C03636=1129.592,11.692,-50.506,179.599,6.524,149.309
C03637=1129.598,11.442,-50.493,179.597,6.519,149.309
C03638=1129.621,10.298,-50.429,179.648,6.418,149.272
C03639=1129.626,10.070,-50.417,179.645,6.416,149.272
C03640=1129.630,9.842,-50.404,179.643,6.415,149.272
C03641=1129.635,9.614,-50.392,179.640,6.415,149.273
C03642=1129.640,9.364,-50.378,179.638,6.414,149.274
C03643=1129.645,9.115,-50.365,179.635,6.413,149.274
C03644=1129.651,8.864,-50.352,179.633,6.412,149.275
C03645=1129.656,8.616,-50.338,179.630,6.411,149.275
C03646=1129.661,8.365,-50.325,179.628,6.411,149.276
C03647=1129.666,8.116,-50.311,179.626,6.409,149.276
C03648=1129.671,7.866,-50.298,179.623,6.409,149.277
C03649=1129.676,7.617,-50.284,179.621,6.408,149.277
C03650=1129.681,7.367,-50.271,179.618,6.406,149.278
C03651=1129.687,7.118,-50.258,179.615,6.406,149.278
C03652=1129.691,6.868,-50.244,179.613,6.405,149.279
C03653=1129.697,6.619,-50.231,179.610,6.403,149.279
C03654=1129.702,6.368,-50.218,179.608,6.403,149.280
C03655=1129.707,6.120,-50.204,179.605,6.402,149.281
C03656=1129.712,5.869,-50.191,179.603,6.401,149.281
C03657=1129.717,5.620,-50.178,179.601,6.400,149.281
C03658=1129.722,5.370,-50.164,179.598,6.399,149.282
C03659=1129.727,5.121,-50.151,179.596,6.399,149.283
C03660=1129.733,4.871,-50.138,179.593,6.397,149.283
C03661=1129.738,4.622,-50.124,179.590,6.397,149.284
C03662=1129.743,4.372,-50.111,179.588,6.396,149.284
C03663=1129.748,4.122,-50.098,179.585,6.394,149.285
C03664=1129.753,3.873,-50.084,179.583,6.394,149.285
C03665=1129.758,3.623,-50.071,179.580,6.393,149.286
C03666=1129.764,3.374,-50.058,179.578,6.392,149.286
C03667=1129.769,3.124,-50.045,179.575,6.391,149.287
C03668=1129.774,2.875,-50.031,179.573,6.390,149.287
C03669=1129.779,2.625,-50.019,179.571,6.389,149.288
C03670=1129.784,2.375,-50.006,179.568,6.388,149.288
C03671=1129.789,2.126,-49.992,179.565,6.387,149.289
C03672=1129.795,1.876,-49.980,179.563,6.386,149.290
C03673=1129.800,1.627,-49.966,179.561,6.386,149.290
C03674=1129.805,1.358,-49.952,179.558,6.384,149.291
C03675=1129.811,1.087,-49.938,179.555,6.384,149.291
C03676=1129.817,0.817,-49.924,179.552,6.382,149.292
C03677=1129.822,0.549,-49.910,179.550,6.382,149.292
C03678=1129.827,0.299,-49.896,179.548,6.381,149.293
C03679=1129.832,0.049,-49.883,179.545,6.380,149.293
C03680=1129.837,-0.201,-49.871,179.542,6.379,149.294
C03681=1129.843,-0.450,-49.857,179.540,6.378,149.294
C03682=1129.848,-0.700,-49.845,179.538,6.378,149.295
C03683=1129.852,-0.950,-49.832,179.535,6.376,149.296
C03684=1129.858,-1.199,-49.819,179.533,6.375,149.296
C03685=1129.863,-1.448,-49.805,179.530,6.375,149.297
C03686=1129.868,-1.698,-49.792,179.528,6.374,149.297
C03687=1129.873,-1.948,-49.779,179.525,6.372,149.298
C03688=1129.878,-2.197,-49.766,179.522,6.372,149.298
C03689=1129.884,-2.447,-49.753,179.520,6.371,149.299
C03690=1129.889,-2.697,-49.740,179.518,6.370,149.299
C03691=1129.894,-2.946,-49.728,179.515,6.369,149.300
C03692=1129.900,-3.195,-49.715,179.513,6.368,149.300
C03693=1129.904,-3.446,-49.702,179.510,6.368,149.301
C03694=1129.910,-3.695,-49.689,179.508,6.367,149.301
C03695=1129.915,-3.944,-49.676,179.505,6.366,149.302
C03696=1129.920,-4.194,-49.663,179.503,6.365,149.303
C03697=1129.925,-4.444,-49.650,179.501,6.364,149.303
C03698=1129.930,-4.693,-49.638,179.498,6.364,149.304
C03699=1129.936,-4.943,-49.624,179.496,6.363,149.304
C03700=1129.941,-5.193,-49.611,179.493,6.361,149.305
C03701=1129.946,-5.442,-49.599,179.491,6.360,149.305
C03702=1129.951,-5.691,-49.586,179.488,6.360,149.306
C03703=1129.957,-5.941,-49.573,179.486,6.359,149.306
C03704=1129.961,-6.192,-49.561,179.483,6.358,149.307
C03705=1129.967,-6.441,-49.548,179.480,6.357,149.307
C03706=1129.972,-6.690,-49.536,179.478,6.356,149.308
C03707=1129.977,-6.940,-49.523,179.476,6.356,149.308
C03708=1129.982,-7.190,-49.509,179.473,6.355,149.309
C03709=1129.987,-7.439,-49.497,179.471,6.354,149.310
C03710=1129.992,-7.689,-49.484,179.468,6.353,149.310
C03711=1129.997,-7.938,-49.472,179.466,6.352,149.310
C03712=1130.002,-8.188,-49.459,179.464,6.352,149.311
C03713=1130.008,-8.438,-49.446,179.461,6.351,149.312
C03714=1130.013,-8.687,-49.434,179.459,6.349,149.312
C03715=1130.018,-8.937,-49.421,179.456,6.349,149.313
C03716=1130.024,-9.186,-49.408,179.454,6.348,149.313
C03717=1130.028,-9.436,-49.395,179.452,6.347,149.314
C03718=1130.033,-9.686,-49.384,179.449,6.347,149.314
C03719=1130.039,-9.936,-49.370,179.446,6.345,149.315
C03720=1130.044,-10.185,-49.358,179.444,6.345,149.315
C03721=1130.050,-10.434,-49.345,179.442,6.344,149.316
C03722=1130.054,-10.684,-49.332,179.439,6.343,149.317
C03723=1130.060,-10.934,-49.320,179.437,6.343,149.317
C03724=1130.065,-11.184,-49.308,179.434,6.341,149.317
C03725=1130.070,-11.433,-49.295,179.432,6.341,149.318
C03726=1130.075,-11.682,-49.282,179.429,6.340,149.319
C03727=1130.080,-11.932,-49.271,179.427,6.339,149.319
C03728=1130.086,-12.183,-49.257,179.425,6.338,149.320
C03729=1130.091,-12.432,-49.244,179.422,6.338,149.320
C03730=1130.096,-12.682,-49.233,179.420,6.336,149.321
C03731=1130.101,-12.931,-49.220,179.417,6.335,149.321
C03732=1130.106,-13.180,-49.207,179.415,6.335,149.322
C03733=1130.112,-13.430,-49.195,179.413,6.334,149.322
C03734=1130.116,-13.680,-49.182,179.410,6.333,149.323
C03735=1130.121,-13.930,-49.170,179.408,6.333,149.324
C03736=1130.127,-14.180,-49.158,179.405,6.331,149.324
C03737=1130.132,-14.429,-49.145,179.403,6.331,149.324
C03738=1130.137,-14.678,-49.133,179.401,6.330,149.325
C03739=1130.143,-14.928,-49.121,179.398,6.329,149.326
C03740=1130.148,-15.177,-49.108,179.396,6.329,149.326
C03741=1130.153,-15.427,-49.096,179.394,6.328,149.327
C03742=1130.158,-15.677,-49.084,179.390,6.327,149.327
C03743=1130.163,-15.927,-49.071,179.388,6.326,149.328
C03744=1130.168,-16.177,-49.059,179.386,6.325,149.328
C03745=1130.173,-16.426,-49.046,179.384,6.324,149.329
C03746=1130.179,-16.676,-49.034,179.381,6.324,149.329
C03747=1130.184,-16.925,-49.022,179.379,6.323,149.330
C03748=1130.189,-17.175,-49.010,179.377,6.322,149.330
C03749=1130.194,-17.425,-48.997,179.373,6.321,149.331
C03750=1130.200,-17.674,-48.985,179.371,6.320,149.331
C03751=1130.205,-17.924,-48.973,179.369,6.320,149.332
C03752=1130.210,-18.173,-48.960,179.366,6.319,149.333
C03753=1130.216,-18.423,-48.948,179.364,6.318,149.333
C03754=1130.221,-18.672,-48.936,179.362,6.318,149.334
C03755=1130.226,-18.922,-48.924,179.360,6.317,149.334
C03756=1130.231,-19.172,-48.911,179.357,6.316,149.335
C03757=1130.237,-19.422,-48.899,179.354,6.315,149.335
C03758=1130.241,-19.671,-48.888,179.352,6.314,149.336
C03759=1130.246,-19.921,-48.875,179.350,6.314,149.336
C03760=1130.251,-20.171,-48.863,179.347,6.313,149.337
C03761=1130.256,-20.420,-48.851,179.345,6.312,149.337
C03762=1130.262,-20.670,-48.839,179.343,6.311,149.338
C03763=1130.267,-20.920,-48.826,179.340,6.311,149.338
C03764=1130.272,-21.170,-48.814,179.338,6.310,149.339
C03765=1130.278,-21.420,-48.802,179.335,6.309,149.339
C03766=1130.283,-21.669,-48.790,179.333,6.308,149.340
C03767=1130.288,-21.919,-48.779,179.331,6.307,149.341
C03768=1130.293,-22.168,-48.766,179.328,6.307,149.341
C03769=1130.298,-22.418,-48.754,179.326,6.306,149.342
C03770=1130.304,-22.668,-48.742,179.323,6.305,149.342
C03771=1130.309,-22.917,-48.730,179.321,6.305,149.343
C03772=1130.315,-23.166,-48.718,179.319,6.304,149.343
C03773=1130.320,-23.416,-48.706,179.316,6.303,149.344
C03774=1130.325,-23.665,-48.694,179.314,6.302,149.344
C03775=1130.330,-23.915,-48.682,179.311,6.301,149.345
C03776=1130.335,-24.165,-48.670,179.309,6.300,149.345
C03777=1130.341,-24.414,-48.658,179.307,6.300,149.346
C03778=1130.346,-24.685,-48.645,179.304,6.299,149.346
C03779=1130.351,-24.955,-48.632,179.302,6.299,149.347
C03780=1130.357,-25.225,-48.619,179.299,6.297,149.348
C03781=1130.362,-25.495,-48.606,179.296,6.297,149.348
C03782=1130.368,-25.745,-48.594,179.294,6.296,149.349
C03783=1130.373,-25.995,-48.583,179.292,6.295,149.349
C03784=1130.379,-26.245,-48.571,179.290,6.294,149.350
C03785=1130.383,-26.494,-48.559,179.287,6.294,149.350
C03786=1130.389,-26.743,-48.547,179.285,6.293,149.351
C03787=1130.395,-26.993,-48.535,179.283,6.292,149.351
C03788=1130.400,-27.243,-48.523,179.280,6.292,149.352
C03789=1130.404,-27.492,-48.511,179.277,6.290,149.353
C03790=1130.410,-27.742,-48.499,179.275,6.290,149.353
C03791=1130.415,-27.992,-48.488,179.273,6.289,149.354
C03792=1130.421,-28.242,-48.476,179.270,6.288,149.354
C03793=1130.425,-28.491,-48.464,179.268,6.288,149.355
C03794=1130.431,-28.741,-48.453,179.266,6.287,149.355
C03795=1130.436,-28.991,-48.440,179.264,6.286,149.356
C03796=1130.441,-29.240,-48.429,179.261,6.286,149.356
C03797=1130.447,-29.490,-48.417,179.259,6.285,149.357
C03798=1130.452,-29.740,-48.405,179.257,6.284,149.357
C03799=1130.457,-29.989,-48.394,179.254,6.284,149.358
C03800=1130.462,-30.239,-48.382,179.252,6.283,149.358
C03801=1130.468,-30.489,-48.370,179.250,6.282,149.359
C03802=1130.472,-30.739,-48.359,179.247,6.281,149.359
C03803=1130.477,-30.988,-48.346,179.245,6.281,149.360
C03804=1130.483,-31.238,-48.334,179.243,6.280,149.361
C03805=1130.488,-31.487,-48.323,179.240,6.280,149.361
C03806=1130.494,-31.737,-48.312,179.237,6.278,149.362
C03807=1130.498,-31.986,-48.300,179.235,6.278,149.362
C03808=1130.504,-32.236,-48.288,179.233,6.277,149.363
C03809=1130.509,-32.486,-48.277,179.231,6.276,149.363
C03810=1130.514,-32.736,-48.265,179.228,6.276,149.364
C03811=1130.520,-32.985,-48.254,179.226,6.275,149.364
C03812=1130.525,-33.235,-48.242,179.224,6.274,149.365
C03813=1130.530,-33.485,-48.231,179.221,6.273,149.365
C03814=1130.535,-33.735,-48.219,179.219,6.273,149.366
C03815=1130.540,-33.984,-48.207,179.216,6.272,149.366
C03816=1130.546,-34.233,-48.196,179.214,6.271,149.367
C03817=1130.551,-34.483,-48.185,179.212,6.271,149.367
C03818=1130.556,-34.733,-48.173,179.209,6.270,149.368
C03819=1130.562,-34.983,-48.161,179.207,6.269,149.369
C03820=1130.566,-35.233,-48.149,179.205,6.269,149.369
C03821=1130.572,-35.482,-48.138,179.202,6.268,149.370
C03822=1130.577,-35.731,-48.127,179.200,6.267,149.370
C03823=1130.583,-35.981,-48.115,179.198,6.267,149.371
C03824=1130.587,-36.231,-48.104,179.196,6.266,149.371
C03825=1130.593,-36.481,-48.092,179.193,6.265,149.372
C03826=1130.598,-36.731,-48.081,179.191,6.265,149.372
C03827=1130.604,-36.980,-48.070,179.189,6.264,149.373
C03828=1130.608,-37.230,-48.058,179.187,6.263,149.373
C03829=1130.614,-37.480,-48.046,179.184,6.263,149.374
C03830=1130.619,-37.729,-48.035,179.182,6.262,149.375
C03831=1130.625,-37.979,-48.024,179.180,6.261,149.375
C03832=1130.629,-38.228,-48.012,179.177,6.260,149.375
C03833=1130.635,-38.478,-48.000,179.175,6.260,149.376
C03834=1130.640,-38.728,-47.990,179.173,6.259,149.377
C03835=1130.646,-38.978,-47.978,179.170,6.258,149.377
C03836=1130.650,-39.228,-47.967,179.168,6.258,149.378
C03837=1130.656,-39.477,-47.955,179.165,6.257,149.378
C03838=1130.661,-39.726,-47.944,179.163,6.257,149.379
C03839=1130.667,-39.976,-47.932,179.161,6.256,149.379
C03840=1130.672,-40.227,-47.922,179.159,6.255,149.380
C03841=1130.678,-40.476,-47.910,179.156,6.255,149.380
C03842=1130.682,-40.725,-47.899,179.154,6.254,149.381
C03843=1130.687,-40.975,-47.888,179.152,6.253,149.381
C03844=1130.693,-41.225,-47.877,179.149,6.253,149.382
C03845=1130.698,-41.475,-47.866,179.147,6.252,149.383
C03846=1130.703,-41.724,-47.854,179.145,6.251,149.383
C03847=1130.708,-41.974,-47.842,179.143,6.250,149.384
C03848=1130.714,-42.224,-47.832,179.140,6.250,149.384
C03849=1130.719,-42.474,-47.820,179.138,6.249,149.385
C03850=1130.724,-42.723,-47.809,179.136,6.248,149.385
C03851=1130.730,-42.972,-47.797,179.133,6.248,149.386
C03852=1130.735,-43.223,-47.787,179.131,6.247,149.386
C03853=1130.740,-43.472,-47.776,179.129,6.246,149.387
C03854=1130.746,-43.722,-47.764,179.126,6.246,149.387
C03855=1130.751,-43.972,-47.753,179.124,6.245,149.388
C03856=1130.755,-44.221,-47.742,179.122,6.245,149.389
C03857=1130.761,-44.471,-47.731,179.119,6.244,149.389
C03858=1130.766,-44.721,-47.720,179.117,6.243,149.389
C03859=1130.771,-44.971,-47.709,179.115,6.242,149.390
C03860=1130.777,-45.220,-47.697,179.113,6.241,149.390
C03861=1130.782,-45.470,-47.687,179.110,6.241,149.391
C03862=1130.787,-45.719,-47.676,179.108,6.240,149.392
C03863=1130.793,-45.969,-47.664,179.106,6.240,149.392
C03864=1130.798,-46.219,-47.653,179.104,6.239,149.393
C03865=1130.803,-46.468,-47.642,179.101,6.238,149.393
C03866=1130.809,-46.719,-47.631,179.099,6.238,149.394
C03867=1130.813,-46.968,-47.620,179.097,6.238,149.394
C03868=1130.819,-47.217,-47.609,179.095,6.237,149.395
C03869=1130.824,-47.468,-47.598,179.092,6.236,149.395
C03870=1130.830,-47.717,-47.587,179.090,6.236,149.396
C03871=1130.835,-47.967,-47.576,179.088,6.235,149.396
C03872=1130.839,-48.217,-47.565,179.086,6.234,149.397
C03873=1130.846,-48.466,-47.554,179.083,6.234,149.398
C03874=1130.850,-48.716,-47.543,179.081,6.233,149.398
C03875=1130.856,-48.966,-47.533,179.079,6.232,149.398
C03876=1130.861,-49.215,-47.521,179.076,6.231,149.399
C03877=1130.867,-49.465,-47.511,179.074,6.231,149.400
C03878=1130.872,-49.715,-47.499,179.072,6.230,149.400
C03879=1130.877,-49.965,-47.489,179.069,6.230,149.401
C03880=1130.882,-50.214,-47.478,179.067,6.229,149.401
C03881=1130.888,-50.464,-47.467,179.065,6.228,149.402
C03882=1130.893,-50.734,-47.455,179.062,6.228,149.402
C03883=1130.899,-51.005,-47.443,179.060,6.227,149.403
C03884=1130.905,-51.276,-47.431,179.057,6.227,149.403
C03885=1130.910,-51.547,-47.420,179.055,6.226,149.404
C03886=1130.916,-51.797,-47.408,179.053,6.225,149.404
C03887=1130.921,-52.046,-47.398,179.050,6.225,149.405
C03888=1130.926,-52.296,-47.387,179.048,6.224,149.406
C03889=1130.932,-52.546,-47.377,179.046,6.223,149.406
C03890=1130.937,-52.796,-47.366,179.044,6.222,149.407
C03891=1130.942,-53.045,-47.355,179.042,6.223,149.407
C03892=1130.948,-53.295,-47.344,179.040,6.222,149.408
C03893=1130.952,-53.545,-47.333,179.037,6.221,149.408
C03894=1130.958,-53.794,-47.323,179.035,6.220,149.409
C03895=1130.963,-54.045,-47.312,179.033,6.220,149.409
C03896=1130.968,-54.294,-47.301,179.030,6.219,149.410
C03897=1130.973,-54.544,-47.291,179.028,6.218,149.410
C03898=1130.979,-54.793,-47.280,179.026,6.218,149.411
C03899=1130.984,-55.043,-47.268,179.024,6.217,149.411
C03900=1130.990,-55.293,-47.258,179.021,6.217,149.412
C03901=1130.995,-55.542,-47.247,179.019,6.216,149.413
C03902=1131.000,-55.792,-47.237,179.017,6.216,149.413
C03903=1131.005,-56.042,-47.226,179.015,6.215,149.413
C03904=1131.011,-56.292,-47.216,179.013,6.214,149.414
C03905=1131.015,-56.541,-47.205,179.010,6.214,149.415
C03906=1131.021,-56.791,-47.194,179.008,6.213,149.415
C03907=1131.026,-57.041,-47.184,179.006,6.212,149.416
C03908=1131.031,-57.290,-47.173,179.004,6.212,149.416
C03909=1131.037,-57.540,-47.163,179.001,6.211,149.417
C03910=1131.042,-57.790,-47.152,178.999,6.210,149.417
C03911=1131.048,-58.039,-47.142,178.997,6.210,149.418
C03912=1131.052,-58.289,-47.131,178.995,6.210,149.418
C03913=1131.058,-58.539,-47.120,178.993,6.209,149.419
C03914=1131.063,-58.789,-47.110,178.990,6.209,149.419
C03915=1131.068,-59.038,-47.100,178.988,6.208,149.420
C03916=1131.073,-59.288,-47.088,178.986,6.207,149.420
C03917=1131.079,-59.538,-47.078,178.984,6.206,149.421
C03918=1131.084,-59.787,-47.068,178.981,6.206,149.421
C03919=1131.089,-60.037,-47.057,178.979,6.206,149.422
C03920=1131.095,-60.287,-47.047,178.977,6.205,149.423
C03921=1131.100,-60.537,-47.036,178.975,6.204,149.423
C03922=1131.105,-60.786,-47.026,178.973,6.204,149.424
C03923=1131.110,-61.036,-47.015,178.971,6.203,149.424
C03924=1131.116,-61.286,-47.005,178.968,6.203,149.425
C03925=1131.121,-61.535,-46.995,178.966,6.202,149.425
C03926=1131.126,-61.786,-46.984,178.963,6.201,149.426
C03927=1131.132,-62.035,-46.973,178.962,6.201,149.426
C03928=1131.137,-62.285,-46.963,178.960,6.200,149.427
C03929=1131.142,-62.534,-46.952,178.957,6.200,149.427
C03930=1131.148,-62.784,-46.942,178.955,6.199,149.428
C03931=1131.153,-63.034,-46.932,178.953,6.198,149.428
C03932=1131.158,-63.284,-46.921,178.950,6.198,149.429
C03933=1131.163,-63.534,-46.911,178.948,6.197,149.429
C03934=1131.169,-63.784,-46.901,178.946,6.197,149.430
C03935=1131.175,-64.033,-46.890,178.944,6.196,149.430
C03936=1131.180,-64.283,-46.880,178.942,6.196,149.431
C03937=1131.185,-64.533,-46.870,178.940,6.195,149.431
C03938=1131.191,-64.782,-46.859,178.937,6.194,149.432
C03939=1131.195,-65.032,-46.849,178.935,6.193,149.432
C03940=1131.200,-65.281,-46.839,178.933,6.194,149.433
C03941=1131.206,-65.531,-46.828,178.931,6.193,149.434
C03942=1131.211,-65.781,-46.818,178.929,6.192,149.434
C03943=1131.217,-66.031,-46.808,178.927,6.192,149.435
C03944=1131.222,-66.280,-46.797,178.924,6.191,149.435
C03945=1131.227,-66.530,-46.787,178.922,6.190,149.436
C03946=1131.233,-66.780,-46.777,178.920,6.190,149.436
C03947=1131.238,-67.029,-46.767,178.918,6.190,149.437
C03948=1131.243,-67.279,-46.756,178.916,6.189,149.437
C03949=1131.248,-67.529,-46.746,178.914,6.188,149.438
C03950=1131.254,-67.778,-46.736,178.911,6.188,149.438
C03951=1131.259,-68.029,-46.725,178.909,6.187,149.439
C03952=1131.264,-68.278,-46.715,178.907,6.187,149.439
C03953=1131.270,-68.528,-46.706,178.905,6.186,149.440
C03954=1131.275,-68.778,-46.696,178.903,6.186,149.440
C03955=1131.280,-69.028,-46.685,178.901,6.185,149.441
C03956=1131.286,-69.277,-46.675,178.898,6.184,149.441
C03957=1131.291,-69.527,-46.665,178.896,6.184,149.442
C03958=1131.296,-69.777,-46.654,178.894,6.184,149.442
C03959=1131.301,-70.026,-46.645,178.892,6.183,149.443
C03960=1131.307,-70.276,-46.635,178.890,6.182,149.443
C03961=1131.312,-70.526,-46.624,178.887,6.181,149.444
C03962=1131.317,-70.776,-46.614,178.885,6.181,149.445
C03963=1131.323,-71.025,-46.604,178.883,6.181,149.445
C03964=1131.328,-71.275,-46.595,178.881,6.180,149.446
C03965=1131.333,-71.525,-46.584,178.879,6.180,149.446
C03966=1131.339,-71.775,-46.574,178.877,6.179,149.447
C03967=1131.344,-72.025,-46.564,178.874,6.178,149.447
C03968=1131.349,-72.274,-46.554,178.872,6.178,149.448
C03969=1131.354,-72.524,-46.544,178.870,6.178,149.448
C03970=1131.360,-72.774,-46.534,178.868,6.177,149.449
C03971=1131.366,-73.024,-46.524,178.866,6.176,149.449
C03972=1131.371,-73.273,-46.514,178.864,6.175,149.450
C03973=1131.376,-73.522,-46.504,178.862,6.175,149.450
C03974=1131.381,-73.773,-46.493,178.859,6.175,149.451
C03975=1131.387,-74.023,-46.484,178.857,6.174,149.451
C03976=1131.392,-74.272,-46.474,178.855,6.174,149.452
C03977=1131.398,-74.522,-46.464,178.853,6.173,149.452
C03978=1131.403,-74.772,-46.454,178.851,6.173,149.453
C03979=1131.407,-75.021,-46.444,178.849,6.172,149.453
C03980=1131.413,-75.271,-46.434,178.847,6.171,149.454
C03981=1131.419,-75.521,-46.424,178.844,6.171,149.454
C03982=1131.425,-75.770,-46.414,178.842,6.170,149.455
C03983=1131.429,-76.021,-46.405,178.840,6.170,149.455
C03984=1131.435,-76.270,-46.395,178.838,6.169,149.456
C03985=1131.440,-76.520,-46.384,178.836,6.169,149.456
C03986=1131.446,-76.792,-46.374,178.833,6.168,149.457
C03987=1131.452,-77.063,-46.364,178.831,6.168,149.458
C03988=1131.458,-77.335,-46.353,178.829,6.167,149.458
C03989=1131.463,-77.606,-46.342,178.826,6.166,149.459
C03990=1131.469,-77.856,-46.332,178.825,6.167,149.459
C03991=1131.475,-78.106,-46.322,178.822,6.166,149.460
C03992=1131.479,-78.355,-46.313,178.820,6.165,149.460
C03993=1131.485,-78.605,-46.302,178.818,6.164,149.461
C03994=1131.490,-78.855,-46.293,178.816,6.164,149.461
C03995=1131.495,-79.105,-46.283,178.814,6.164,149.462
C03996=1131.501,-79.354,-46.273,178.812,6.163,149.462
C03997=1131.506,-79.604,-46.264,178.809,6.162,149.463
C03998=1131.511,-79.854,-46.254,178.808,6.162,149.463
C03999=1131.517,-80.103,-46.245,178.806,6.162,149.464
C04000=1131.522,-80.353,-46.234,178.803,6.161,149.464
C04001=1131.527,-80.603,-46.224,178.801,6.160,149.465
C04002=1131.532,-80.853,-46.215,178.800,6.160,149.465
C04003=1131.538,-81.103,-46.205,178.797,6.159,149.466
C04004=1131.543,-81.352,-46.196,178.795,6.159,149.466
C04005=1131.549,-81.602,-46.186,178.793,6.158,149.467
C04006=1131.554,-81.851,-46.176,178.791,6.158,149.467
C04007=1131.560,-82.101,-46.167,178.789,6.158,149.468
C04008=1131.565,-82.351,-46.156,178.787,6.157,149.468
C04009=1131.570,-82.601,-46.147,178.784,6.156,149.469
C04010=1131.575,-82.851,-46.137,178.783,6.156,149.469
C04011=1131.580,-83.101,-46.128,178.780,6.156,149.470
C04012=1131.586,-83.350,-46.118,178.778,6.155,149.471
C04013=1131.591,-83.600,-46.109,178.776,6.154,149.471
C04014=1131.597,-83.850,-46.099,178.774,6.154,149.472
C04015=1131.602,-84.100,-46.090,178.772,6.154,149.472
C04016=1131.608,-84.349,-46.080,178.770,6.153,149.472
C04017=1131.613,-84.599,-46.071,178.767,6.152,149.473
C04018=1131.618,-84.849,-46.060,178.766,6.152,149.473
C04019=1131.624,-85.098,-46.052,178.764,6.151,149.474
C04020=1131.629,-85.348,-46.041,178.761,6.151,149.475
C04021=1131.634,-85.599,-46.032,178.759,6.151,149.475
C04022=1131.639,-85.848,-46.022,178.757,6.150,149.476
C04023=1131.644,-86.098,-46.013,178.755,6.150,149.476
C04024=1131.650,-86.348,-46.003,178.753,6.149,149.477
C04025=1131.655,-86.597,-45.994,178.751,6.149,149.477
C04026=1131.661,-86.848,-45.984,178.749,6.148,149.478
C04027=1131.666,-87.097,-45.975,178.747,6.147,149.478
C04028=1131.671,-87.347,-45.966,178.745,6.147,149.479
C04029=1131.677,-87.596,-45.956,178.743,6.147,149.479
C04030=1131.682,-87.846,-45.947,178.740,6.146,149.480
C04031=1131.688,-88.096,-45.936,178.738,6.145,149.480
C04032=1131.693,-88.345,-45.928,178.737,6.145,149.481
C04033=1131.699,-88.596,-45.918,178.734,6.145,149.481
C04034=1131.703,-88.845,-45.908,178.732,6.144,149.482
C04035=1131.709,-89.095,-45.900,178.730,6.143,149.482
C04036=1131.715,-89.345,-45.890,178.728,6.143,149.483
C04037=1131.719,-89.594,-45.880,178.726,6.143,149.483
C04038=1131.725,-89.844,-45.871,178.724,6.142,149.484
C04039=1131.730,-90.094,-45.862,178.722,6.142,149.484
C04040=1131.735,-90.343,-45.852,178.720,6.141,149.485
C04041=1131.741,-90.593,-45.843,178.718,6.141,149.485
C04042=1131.746,-90.843,-45.834,178.716,6.141,149.486
C04043=1131.751,-91.093,-45.824,178.714,6.140,149.486
C04044=1131.757,-91.343,-45.815,178.712,6.139,149.487
C04045=1131.762,-91.593,-45.806,178.709,6.138,149.487
C04046=1131.768,-91.842,-45.796,178.708,6.139,149.488
C04047=1131.773,-92.092,-45.787,178.706,6.138,149.488
C04048=1131.778,-92.342,-45.778,178.703,6.137,149.489
C04049=1131.784,-92.591,-45.768,178.702,6.137,149.489
C04050=1131.789,-92.841,-45.759,178.700,6.136,149.490
C04051=1131.794,-93.091,-45.750,178.697,6.136,149.490
C04052=1131.800,-93.341,-45.741,178.695,6.136,149.491
C04053=1131.805,-93.590,-45.731,178.693,6.135,149.491
C04054=1131.810,-93.840,-45.722,178.691,6.135,149.492
C04055=1131.816,-94.090,-45.713,178.689,6.135,149.492
C04056=1131.821,-94.340,-45.704,178.687,6.134,149.493
C04057=1131.826,-94.590,-45.695,178.685,6.133,149.493
C04058=1131.832,-94.840,-45.685,178.683,6.133,149.494
C04059=1131.837,-95.090,-45.676,178.681,6.132,149.494
C04060=1131.842,-95.339,-45.667,178.679,6.132,149.495
C04061=1131.847,-95.589,-45.658,178.677,6.132,149.495
C04062=1131.854,-95.839,-45.649,178.675,6.131,149.496
C04063=1131.859,-96.088,-45.639,178.673,6.130,149.496
C04064=1131.864,-96.338,-45.630,178.671,6.130,149.497
C04065=1131.870,-96.588,-45.621,178.669,6.130,149.497
C04066=1131.875,-96.838,-45.612,178.667,6.129,149.498
C04067=1131.880,-97.088,-45.603,178.665,6.129,149.498
C04068=1131.885,-97.337,-45.594,178.663,6.128,149.499
C04069=1131.891,-97.587,-45.584,178.661,6.128,149.499
C04070=1131.896,-97.837,-45.575,178.659,6.128,149.500
C04071=1131.901,-98.087,-45.566,178.657,6.127,149.500
C04072=1131.906,-98.337,-45.557,178.655,6.126,149.501
C04073=1131.913,-98.586,-45.548,178.653,6.126,149.501
C04074=1131.918,-98.836,-45.539,178.651,6.125,149.502
C04075=1131.923,-99.086,-45.530,178.649,6.125,149.502
C04076=1131.928,-99.336,-45.521,178.647,6.125,149.503
C04077=1131.933,-99.585,-45.512,178.645,6.124,149.503
C04078=1131.939,-99.835,-45.502,178.643,6.123,149.504
C04079=1131.944,-100.085,-45.493,178.641,6.123,149.504
C04080=1131.950,-100.335,-45.484,178.639,6.123,149.505
C04081=1131.955,-100.584,-45.476,178.637,6.122,149.505
C04082=1131.961,-100.834,-45.467,178.635,6.122,149.506
C04083=1131.966,-101.084,-45.458,178.633,6.121,149.506
C04084=1131.972,-101.334,-45.449,178.631,6.120,149.507
C04085=1131.977,-101.584,-45.440,178.629,6.121,149.507
C04086=1131.982,-101.833,-45.431,178.626,6.120,149.508
C04087=1131.987,-102.083,-45.422,178.625,6.120,149.508
C04088=1131.993,-102.332,-45.413,178.623,6.119,149.509
C04089=1131.999,-102.583,-45.404,178.620,6.119,149.509
C04090=1132.005,-102.855,-45.394,178.618,6.118,149.510
C04091=1132.010,-103.127,-45.384,178.617,6.118,149.510
C04092=1132.016,-103.400,-45.375,178.614,6.117,149.511
C04093=1132.022,-103.672,-45.365,178.612,6.117,149.511
C04094=1132.027,-103.922,-45.356,178.609,6.116,149.512
C04095=1132.033,-104.171,-45.348,178.608,6.116,149.512
C04096=1132.038,-104.421,-45.339,178.606,6.115,149.513
C04097=1132.043,-104.671,-45.330,178.604,6.115,149.513
C04098=1132.048,-104.921,-45.321,178.602,6.115,149.514
C04099=1132.054,-105.171,-45.312,178.600,6.114,149.514
C04100=1132.059,-105.421,-45.303,178.598,6.114,149.515
C04101=1132.065,-105.670,-45.294,178.596,6.113,149.515
C04102=1132.070,-105.920,-45.285,178.594,6.113,149.516
C04103=1132.075,-106.170,-45.276,178.592,6.112,149.516
C04104=1132.080,-106.419,-45.267,178.590,6.112,149.517
C04105=1132.086,-106.669,-45.258,178.588,6.112,149.517
C04106=1132.091,-106.918,-45.250,178.586,6.111,149.518
C04107=1132.097,-107.169,-45.242,178.584,6.110,149.518
C04108=1132.102,-107.419,-45.233,178.582,6.110,149.519
C04109=1132.107,-107.669,-45.224,178.580,6.110,149.519
C04110=1132.113,-107.918,-45.215,178.579,6.110,149.520
C04111=1132.118,-108.168,-45.207,178.576,6.109,149.520
C04112=1132.123,-108.417,-45.198,178.574,6.108,149.521
C04113=1132.128,-108.667,-45.189,178.573,6.108,149.521
C04114=1132.135,-108.918,-45.180,178.570,6.107,149.522
C04115=1132.140,-109.167,-45.171,178.569,6.107,149.522
C04116=1132.146,-109.417,-45.163,178.567,6.107,149.523
C04117=1132.151,-109.667,-45.154,178.564,6.106,149.523
C04118=1132.156,-109.917,-45.145,178.563,6.106,149.524
C04119=1132.162,-110.166,-45.136,178.561,6.105,149.524
C04120=1132.167,-110.416,-45.128,178.559,6.105,149.525
C04121=1132.172,-110.666,-45.119,178.557,6.105,149.525
C04122=1132.178,-110.915,-45.111,178.555,6.104,149.526
C04123=1132.183,-111.165,-45.102,178.553,6.104,149.526
C04124=1132.188,-111.415,-45.093,178.551,6.103,149.527
C04125=1132.194,-111.666,-45.085,178.549,6.103,149.527
C04126=1132.200,-111.915,-45.076,178.547,6.102,149.528
C04127=1132.205,-112.165,-45.067,178.545,6.102,149.528
C04128=1132.210,-112.414,-45.058,178.543,6.102,149.528
C04129=1132.215,-112.665,-45.050,178.541,6.101,149.529
C04130=1132.220,-112.914,-45.042,178.539,6.101,149.529
C04131=1132.226,-113.164,-45.033,178.537,6.100,149.530
C04132=1132.231,-113.413,-45.024,178.536,6.100,149.530
C04133=1132.237,-113.663,-45.017,178.533,6.100,149.531
C04134=1132.242,-113.913,-45.008,178.531,6.099,149.531
C04135=1132.247,-114.163,-44.999,178.530,6.099,149.532
C04136=1132.253,-114.412,-44.990,178.528,6.098,149.532
C04137=1132.258,-114.663,-44.982,178.526,6.098,149.533
C04138=1132.264,-114.912,-44.973,178.524,6.097,149.533
C04139=1132.269,-115.162,-44.965,178.522,6.096,149.534
C04140=1132.275,-115.412,-44.956,178.520,6.096,149.534
C04141=1132.280,-115.662,-44.948,178.518,6.096,149.535
C04142=1132.285,-115.912,-44.939,178.516,6.096,149.535
C04143=1132.291,-116.161,-44.931,178.514,6.095,149.536
C04144=1132.296,-116.411,-44.922,178.513,6.095,149.536
C04145=1132.301,-116.660,-44.914,178.510,6.094,149.537
C04146=1132.307,-116.911,-44.906,178.509,6.094,149.537
C04147=1132.312,-117.160,-44.897,178.507,6.094,149.538
C04148=1132.318,-117.410,-44.888,178.504,6.093,149.538
C04149=1132.323,-117.660,-44.880,178.503,6.093,149.538
C04150=1132.329,-117.910,-44.871,178.501,6.092,149.539
C04151=1132.335,-118.160,-44.863,178.499,6.092,149.539
C04152=1132.340,-118.410,-44.855,178.497,6.091,149.540
C04153=1132.344,-118.659,-44.846,178.495,6.091,149.540
C04154=1132.350,-118.909,-44.838,178.493,6.091,149.541
C04155=1132.355,-119.159,-44.830,178.491,6.090,149.541
C04156=1132.361,-119.409,-44.821,178.489,6.090,149.542
C04157=1132.367,-119.658,-44.813,178.487,6.089,149.542
C04158=1132.372,-119.908,-44.804,178.486,6.089,149.543
C04159=1132.377,-120.158,-44.797,178.484,6.088,149.543
C04160=1132.382,-120.408,-44.788,178.482,6.088,149.544
C04161=1132.388,-120.658,-44.780,178.480,6.088,149.544
C04162=1132.394,-120.907,-44.771,178.478,6.088,149.545
C04163=1132.399,-121.158,-44.763,178.476,6.087,149.545
C04164=1132.404,-121.407,-44.754,178.475,6.087,149.546
C04165=1132.410,-121.657,-44.747,178.472,6.086,149.546
C04166=1132.415,-121.907,-44.738,178.470,6.085,149.547
C04167=1132.421,-122.157,-44.730,178.469,6.085,149.547
C04168=1132.426,-122.406,-44.721,178.466,6.085,149.548
C04169=1132.431,-122.657,-44.713,178.465,6.085,149.548
C04170=1132.436,-122.906,-44.705,178.463,6.084,149.549
C04171=1132.442,-123.156,-44.697,178.461,6.084,149.549
C04172=1132.448,-123.405,-44.688,178.459,6.083,149.549
C04173=1132.453,-123.656,-44.680,178.458,6.083,149.550
C04174=1132.458,-123.905,-44.672,178.456,6.082,149.550
C04175=1132.464,-124.155,-44.664,178.454,6.082,149.551
C04176=1132.469,-124.405,-44.655,178.452,6.082,149.551
C04177=1132.475,-124.655,-44.647,178.450,6.082,149.552
C04178=1132.479,-124.904,-44.639,178.448,6.081,149.552
C04179=1132.485,-125.154,-44.631,178.446,6.081,149.553
C04180=1132.491,-125.404,-44.622,178.444,6.080,149.553
C04181=1132.497,-125.654,-44.615,178.443,6.080,149.554
C04182=1132.501,-125.904,-44.607,178.440,6.079,149.554
C04183=1132.507,-126.154,-44.598,178.438,6.079,149.555
C04184=1132.513,-126.403,-44.590,178.437,6.078,149.555
C04185=1132.517,-126.653,-44.582,178.435,6.078,149.555
C04186=1132.523,-126.903,-44.574,178.433,6.078,149.556
C04187=1132.529,-127.153,-44.566,178.431,6.077,149.556
C04188=1132.534,-127.402,-44.557,178.429,6.077,149.557
C04189=1132.539,-127.653,-44.550,178.427,6.076,149.557
C04190=1132.545,-127.902,-44.541,178.426,6.076,149.558
C04191=1132.550,-128.152,-44.533,178.423,6.076,149.558
C04192=1132.556,-128.402,-44.526,178.422,6.076,149.559
C04193=1132.561,-128.651,-44.517,178.420,6.075,149.559
C04194=1132.140,-128.663,-44.562,178.417,6.079,149.561
C04195=1132.135,-128.413,-44.570,178.418,6.079,149.560
C04196=1132.129,-128.163,-44.577,178.421,6.079,149.560
C04197=1132.124,-127.913,-44.586,178.422,6.079,149.559
C04198=1132.118,-127.664,-44.594,178.424,6.080,149.559
C04199=1132.113,-127.413,-44.602,178.426,6.080,149.559
C04200=1132.108,-127.164,-44.610,178.428,6.081,149.558
C04201=1132.102,-126.914,-44.618,178.429,6.081,149.558
C04202=1132.097,-126.665,-44.626,178.432,6.082,149.557
C04203=1132.092,-126.415,-44.634,178.434,6.082,149.557
C04204=1132.086,-126.164,-44.643,178.435,6.082,149.556
C04205=1132.080,-125.915,-44.651,178.438,6.083,149.556
C04206=1132.076,-125.665,-44.659,178.439,6.083,149.555
C04207=1132.070,-125.416,-44.667,178.441,6.084,149.555
C04208=1132.064,-125.165,-44.675,178.443,6.084,149.554
C04209=1132.059,-124.916,-44.683,178.445,6.085,149.554
C04210=1132.054,-124.666,-44.691,178.446,6.085,149.554
C04211=1132.048,-124.416,-44.699,178.449,6.086,149.553
C04212=1132.043,-124.166,-44.708,178.450,6.086,149.553
C04213=1132.038,-123.916,-44.716,178.452,6.086,149.552
C04214=1132.032,-123.667,-44.724,178.454,6.086,149.552
C04215=1132.027,-123.416,-44.733,178.456,6.087,149.551
C04216=1132.021,-123.167,-44.741,178.458,6.087,149.551
C04217=1132.015,-122.917,-44.749,178.460,6.088,149.550
C04218=1132.010,-122.668,-44.757,178.461,6.088,149.550
C04219=1132.005,-122.418,-44.765,178.463,6.089,149.549
C04220=1132.000,-122.168,-44.774,178.465,6.090,149.549
C04221=1131.994,-121.918,-44.782,178.467,6.089,149.548
C04222=1131.989,-121.668,-44.790,178.469,6.090,149.548
C04223=1131.983,-121.419,-44.798,178.471,6.090,149.547
C04224=1131.978,-121.169,-44.807,178.473,6.091,149.547
C04225=1131.972,-120.918,-44.815,178.475,6.091,149.546
C04226=1131.967,-120.669,-44.824,178.477,6.092,149.546
C04227=1131.962,-120.419,-44.831,178.478,6.092,149.545
C04228=1131.957,-120.169,-44.840,178.481,6.092,149.545
C04229=1131.951,-119.920,-44.849,178.482,6.092,149.544
C04230=1131.946,-119.669,-44.857,178.484,6.093,149.544
C04231=1131.940,-119.420,-44.866,178.487,6.094,149.543
C04232=1131.934,-119.170,-44.874,178.488,6.094,149.543
C04233=1131.930,-118.920,-44.882,178.490,6.095,149.543
C04234=1131.924,-118.671,-44.890,178.491,6.095,149.542
C04235=1131.919,-118.421,-44.899,178.494,6.096,149.542
C04236=1131.914,-118.171,-44.908,178.495,6.095,149.541
C04237=1131.907,-117.921,-44.915,178.497,6.096,149.541
C04238=1131.902,-117.671,-44.924,178.499,6.096,149.540
C04239=1131.897,-117.421,-44.933,178.501,6.097,149.540
C04240=1131.891,-117.172,-44.941,178.503,6.098,149.539
C04241=1131.887,-116.922,-44.949,178.505,6.098,149.539
C04242=1131.881,-116.672,-44.957,178.507,6.098,149.538
C04243=1131.875,-116.422,-44.966,178.509,6.098,149.538
C04244=1131.870,-116.173,-44.975,178.511,6.099,149.537
C04245=1131.864,-115.923,-44.983,178.513,6.099,149.537
C04246=1131.859,-115.673,-44.992,178.515,6.100,149.536
C04247=1131.854,-115.423,-45.001,178.516,6.100,149.536
C04248=1131.848,-115.173,-45.008,178.519,6.100,149.535
C04249=1131.843,-114.923,-45.017,178.521,6.101,149.535
C04250=1131.837,-114.674,-45.026,178.522,6.101,149.534
C04251=1131.832,-114.423,-45.034,178.525,6.102,149.534
C04252=1131.827,-114.174,-45.042,178.526,6.102,149.533
C04253=1131.822,-113.924,-45.051,178.528,6.103,149.533
C04254=1131.817,-113.675,-45.060,178.531,6.103,149.532
C04255=1131.810,-113.425,-45.068,178.532,6.103,149.532
C04256=1131.805,-113.175,-45.077,178.534,6.104,149.532
C04257=1131.800,-112.925,-45.086,178.536,6.104,149.531
C04258=1131.794,-112.676,-45.094,178.538,6.105,149.531
C04259=1131.789,-112.426,-45.102,178.539,6.105,149.530
C04260=1131.784,-112.176,-45.111,178.542,6.106,149.530
C04261=1131.779,-111.926,-45.120,178.544,6.107,149.529
C04262=1131.773,-111.677,-45.129,178.545,6.106,149.529
C04263=1131.767,-111.426,-45.137,178.548,6.107,149.528
C04264=1131.762,-111.176,-45.146,178.549,6.107,149.528
C04265=1131.756,-110.927,-45.154,178.551,6.108,149.527
C04266=1131.751,-110.677,-45.163,178.554,6.109,149.527
C04267=1131.746,-110.428,-45.172,178.555,6.109,149.526
C04268=1131.741,-110.177,-45.180,178.557,6.109,149.526
C04269=1131.735,-109.928,-45.189,178.559,6.109,149.525
C04270=1131.730,-109.678,-45.198,178.561,6.110,149.525
C04271=1131.724,-109.428,-45.207,178.563,6.111,149.524
C04272=1131.719,-109.178,-45.216,178.565,6.111,149.524
C04273=1131.713,-108.929,-45.223,178.567,6.112,149.523
C04274=1131.708,-108.679,-45.232,178.569,6.111,149.523
C04275=1131.703,-108.429,-45.241,178.571,6.112,149.523
C04276=1131.698,-108.179,-45.250,178.573,6.113,149.522
C04277=1131.692,-107.930,-45.259,178.575,6.113,149.522
C04278=1131.687,-107.680,-45.268,178.577,6.114,149.521
C04279=1131.682,-107.430,-45.276,178.578,6.114,149.521
C04280=1131.676,-107.180,-45.285,178.581,6.114,149.520
C04281=1131.670,-106.930,-45.294,178.583,6.115,149.520
C04282=1131.665,-106.680,-45.303,178.584,6.115,149.519
C04283=1131.659,-106.431,-45.312,178.587,6.116,149.519
C04284=1131.654,-106.181,-45.320,178.588,6.116,149.518
C04285=1131.649,-105.931,-45.329,178.590,6.116,149.518
C04286=1131.644,-105.681,-45.338,178.593,6.117,149.517
C04287=1131.638,-105.432,-45.347,178.594,6.117,149.517
C04288=1131.633,-105.182,-45.356,178.596,6.118,149.516
C04289=1131.628,-104.932,-45.365,178.599,6.119,149.516
C04290=1131.623,-104.682,-45.373,178.600,6.119,149.515
C04291=1131.617,-104.432,-45.382,178.602,6.119,149.515
C04292=1131.612,-104.183,-45.391,178.604,6.119,149.514
C04293=1131.606,-103.933,-45.400,178.606,6.120,149.514
C04294=1131.601,-103.683,-45.409,178.608,6.121,149.513
C04295=1131.595,-103.411,-45.419,178.611,6.121,149.513
C04296=1131.589,-103.138,-45.428,178.613,6.121,149.512
C04297=1131.583,-102.866,-45.438,178.615,6.122,149.512
C04298=1131.578,-102.594,-45.448,178.617,6.123,149.511
C04299=1131.572,-102.345,-45.457,178.619,6.123,149.511
C04300=1131.567,-102.095,-45.465,178.621,6.123,149.510
C04301=1131.562,-101.845,-45.474,178.623,6.124,149.510
C04302=1131.556,-101.595,-45.484,178.625,6.124,149.509
C04303=1131.551,-101.345,-45.493,178.627,6.125,149.509
C04304=1131.545,-101.095,-45.502,178.629,6.126,149.508
C04305=1131.540,-100.845,-45.511,178.631,6.125,149.508
C04306=1131.534,-100.596,-45.519,178.633,6.126,149.507
C04307=1131.529,-100.346,-45.528,178.636,6.127,149.506
C04308=1131.523,-100.096,-45.537,178.637,6.127,149.506
C04309=1131.518,-99.846,-45.546,178.639,6.127,149.506
C04310=1131.513,-99.596,-45.555,178.642,6.128,149.505
C04311=1131.508,-99.346,-45.564,178.643,6.128,149.505
C04312=1131.502,-99.096,-45.574,178.645,6.129,149.504
C04313=1131.496,-98.848,-45.583,178.648,6.129,149.504
C04314=1131.491,-98.598,-45.592,178.649,6.129,149.503
C04315=1131.486,-98.348,-45.601,178.651,6.130,149.503
C04316=1131.481,-98.098,-45.610,178.654,6.131,149.502
C04317=1131.475,-97.848,-45.619,178.655,6.131,149.502
C04318=1131.470,-97.598,-45.628,178.657,6.132,149.501
C04319=1131.465,-97.348,-45.637,178.660,6.132,149.501
C04320=1131.460,-97.098,-45.646,178.661,6.132,149.500
C04321=1131.454,-96.849,-45.656,178.663,6.133,149.500
C04322=1131.449,-96.599,-45.665,178.666,6.134,149.499
C04323=1131.443,-96.350,-45.673,178.667,6.134,149.499
C04324=1131.437,-96.100,-45.683,178.669,6.135,149.498
C04325=1131.432,-95.850,-45.692,178.672,6.135,149.498
C04326=1131.427,-95.600,-45.701,178.674,6.135,149.497
C04327=1131.422,-95.351,-45.710,178.676,6.136,149.497
C04328=1131.416,-95.101,-45.720,178.678,6.136,149.496
C04329=1131.411,-94.851,-45.729,178.680,6.136,149.496
C04330=1131.406,-94.601,-45.738,178.682,6.137,149.495
C04331=1131.400,-94.351,-45.747,178.684,6.138,149.495
C04332=1131.395,-94.102,-45.757,178.686,6.138,149.494
C04333=1131.390,-93.852,-45.766,178.688,6.139,149.494
C04334=1131.384,-93.602,-45.775,178.690,6.139,149.493
C04335=1131.379,-93.352,-45.784,178.692,6.139,149.493
C04336=1131.374,-93.102,-45.794,178.694,6.140,149.492
C04337=1131.368,-92.852,-45.803,178.696,6.141,149.492
C04338=1131.363,-92.602,-45.812,178.698,6.141,149.491
C04339=1131.358,-92.353,-45.821,178.700,6.141,149.491
C04340=1131.352,-92.103,-45.831,178.702,6.142,149.490
C04341=1131.347,-91.853,-45.840,178.704,6.142,149.490
C04342=1131.342,-91.603,-45.849,178.706,6.143,149.489
C04343=1131.336,-91.354,-45.859,178.708,6.143,149.489
C04344=1131.331,-91.104,-45.868,178.711,6.144,149.488
C04345=1131.326,-90.854,-45.877,178.712,6.144,149.488
C04346=1131.320,-90.604,-45.886,178.714,6.145,149.487
C04347=1131.315,-90.355,-45.896,178.717,6.145,149.487
C04348=1131.310,-90.105,-45.905,178.718,6.145,149.486
C04349=1131.304,-89.855,-45.914,178.720,6.146,149.486
C04350=1131.299,-89.605,-45.924,178.723,6.147,149.485
C04351=1131.293,-89.355,-45.934,178.724,6.147,149.485
C04352=1131.288,-89.106,-45.943,178.727,6.147,149.484
C04353=1131.283,-88.856,-45.952,178.729,6.148,149.483
C04354=1131.277,-88.606,-45.962,178.731,6.149,149.483
C04355=1131.272,-88.357,-45.971,178.733,6.149,149.483
C04356=1131.266,-88.107,-45.981,178.735,6.149,149.482
C04357=1131.261,-87.857,-45.990,178.737,6.150,149.482
C04358=1131.256,-87.607,-46.000,178.739,6.150,149.481
C04359=1131.251,-87.357,-46.009,178.741,6.151,149.481
C04360=1131.246,-87.108,-46.018,178.743,6.152,149.480
C04361=1131.240,-86.858,-46.028,178.745,6.152,149.480
C04362=1131.235,-86.609,-46.037,178.747,6.152,149.479
C04363=1131.229,-86.359,-46.047,178.750,6.153,149.478
C04364=1131.224,-86.109,-46.056,178.752,6.154,149.478
C04365=1131.218,-85.859,-46.066,178.753,6.154,149.477
C04366=1131.213,-85.609,-46.075,178.756,6.154,149.477
C04367=1131.207,-85.360,-46.085,178.758,6.155,149.476
C04368=1131.202,-85.110,-46.094,178.760,6.156,149.476
C04369=1131.197,-84.860,-46.104,178.762,6.156,149.475
C04370=1131.192,-84.611,-46.113,178.764,6.156,149.475
C04371=1131.187,-84.360,-46.124,178.766,6.157,149.474
C04372=1131.181,-84.110,-46.133,178.769,6.158,149.474
C04373=1131.176,-83.861,-46.143,178.770,6.158,149.473
C04374=1131.171,-83.611,-46.152,178.772,6.158,149.473
C04375=1131.165,-83.362,-46.162,178.775,6.159,149.472
C04376=1131.160,-83.112,-46.171,178.777,6.160,149.472
C04377=1131.154,-82.862,-46.181,178.778,6.160,149.471
C04378=1131.149,-82.612,-46.190,178.781,6.161,149.471
C04379=1131.143,-82.363,-46.200,178.783,6.161,149.470
C04380=1131.138,-82.113,-46.209,178.785,6.161,149.470
C04381=1131.133,-81.863,-46.220,178.787,6.162,149.469
C04382=1131.128,-81.613,-46.229,178.789,6.162,149.469
C04383=1131.123,-81.363,-46.239,178.791,6.163,149.468
C04384=1131.117,-81.114,-46.249,178.793,6.163,149.468
C04385=1131.112,-80.864,-46.258,178.795,6.164,149.467
C04386=1131.106,-80.614,-46.268,178.797,6.165,149.467
C04387=1131.101,-80.364,-46.277,178.800,6.165,149.466
C04388=1131.095,-80.115,-46.287,178.802,6.166,149.466
C04389=1131.091,-79.865,-46.297,178.804,6.166,149.465
C04390=1131.085,-79.615,-46.307,178.806,6.166,149.465
C04391=1131.080,-79.365,-46.317,178.808,6.167,149.464
C04392=1131.075,-79.116,-46.326,178.811,6.168,149.464
C04393=1131.069,-78.866,-46.336,178.812,6.168,149.463
C04394=1131.063,-78.616,-46.346,178.814,6.169,149.463
C04395=1131.058,-78.367,-46.355,178.817,6.169,149.462
C04396=1131.053,-78.116,-46.366,178.819,6.170,149.462
C04397=1131.048,-77.867,-46.375,178.821,6.170,149.461
C04398=1131.042,-77.617,-46.385,178.823,6.171,149.461
C04399=1131.036,-77.345,-46.396,178.825,6.171,149.460
C04400=1131.030,-77.074,-46.406,178.828,6.172,149.459
C04401=1131.025,-76.803,-46.417,178.830,6.172,149.459
C04402=1131.019,-76.531,-46.428,178.832,6.173,149.458
C04403=1131.014,-76.281,-46.437,178.834,6.174,149.458
C04404=1131.008,-76.032,-46.448,178.836,6.173,149.457
C04405=1131.003,-75.782,-46.458,178.839,6.174,149.457
C04406=1130.998,-75.532,-46.467,178.841,6.175,149.456
C04407=1130.993,-75.282,-46.477,178.843,6.176,149.456
C04408=1130.987,-75.033,-46.488,178.845,6.176,149.455
C04409=1130.982,-74.783,-46.498,178.847,6.176,149.455
C04410=1130.976,-74.533,-46.507,178.849,6.177,149.454
C04411=1130.971,-74.284,-46.517,178.852,6.178,149.454
C04412=1130.966,-74.033,-46.527,178.854,6.178,149.453
C04413=1130.961,-73.784,-46.537,178.856,6.179,149.453
C04414=1130.955,-73.534,-46.547,178.858,6.179,149.452
C04415=1130.949,-73.284,-46.557,178.860,6.180,149.452
C04416=1130.944,-73.034,-46.567,178.862,6.181,149.451
C04417=1130.940,-72.785,-46.577,178.864,6.181,149.451
C04418=1130.934,-72.535,-46.587,178.866,6.181,149.450
C04419=1130.928,-72.286,-46.597,178.869,6.182,149.450
C04420=1130.923,-72.035,-46.607,178.871,6.182,149.449
C04421=1130.918,-71.786,-46.617,178.873,6.183,149.449
C04422=1130.913,-71.536,-46.627,178.875,6.184,149.448
C04423=1130.907,-71.287,-46.637,178.877,6.185,149.448
C04424=1130.902,-71.036,-46.648,178.879,6.184,149.447
C04425=1130.897,-70.787,-46.657,178.882,6.185,149.446
C04426=1130.891,-70.537,-46.667,178.884,6.186,149.446
C04427=1130.886,-70.288,-46.677,178.886,6.187,149.445
C04428=1130.881,-70.037,-46.688,178.888,6.187,149.445
C04429=1130.875,-69.788,-46.698,178.890,6.187,149.444
C04430=1130.870,-69.538,-46.707,178.892,6.188,149.444
C04431=1130.865,-69.289,-46.718,178.895,6.188,149.443
C04432=1130.860,-69.039,-46.728,178.897,6.189,149.443
C04433=1130.854,-68.789,-46.738,178.899,6.190,149.442
C04434=1130.848,-68.540,-46.749,178.901,6.190,149.442
C04435=1130.843,-68.289,-46.759,178.903,6.191,149.441
C04436=1130.838,-68.040,-46.769,178.905,6.191,149.441
C04437=1130.833,-67.791,-46.779,178.908,6.192,149.440
C04438=1130.828,-67.540,-46.790,178.910,6.193,149.440
C04439=1130.822,-67.291,-46.800,178.912,6.193,149.439
C04440=1130.817,-67.041,-46.810,178.914,6.193,149.439
C04441=1130.811,-66.791,-46.820,178.916,6.194,149.438
C04442=1130.807,-66.541,-46.830,178.919,6.194,149.438
C04443=1130.801,-66.292,-46.840,178.921,6.195,149.437
C04444=1130.795,-66.042,-46.850,178.923,6.196,149.437
C04445=1130.791,-65.792,-46.861,178.925,6.197,149.436
C04446=1130.785,-65.543,-46.871,178.927,6.197,149.436
C04447=1130.780,-65.293,-46.882,178.929,6.197,149.435
C04448=1130.774,-65.043,-46.892,178.932,6.198,149.434
C04449=1130.769,-64.794,-46.902,178.934,6.199,149.434
C04450=1130.764,-64.543,-46.913,178.936,6.199,149.433
C04451=1130.759,-64.294,-46.923,178.938,6.200,149.433
C04452=1130.753,-64.045,-46.933,178.941,6.200,149.432
C04453=1130.748,-63.794,-46.943,178.942,6.200,149.432
C04454=1130.743,-63.545,-46.954,178.945,6.201,149.431
C04455=1130.737,-63.295,-46.964,178.947,6.202,149.431
C04456=1130.732,-63.045,-46.974,178.949,6.203,149.430
C04457=1130.727,-62.795,-46.985,178.952,6.203,149.430
C04458=1130.722,-62.545,-46.995,178.954,6.204,149.429
C04459=1130.716,-62.296,-47.005,178.956,6.205,149.429
C04460=1130.711,-62.047,-47.016,178.958,6.205,149.428
C04461=1130.706,-61.796,-47.027,178.960,6.205,149.428
C04462=1130.700,-61.547,-47.037,178.962,6.206,149.427
C04463=1130.695,-61.297,-47.048,178.965,6.207,149.427
C04464=1130.690,-61.047,-47.058,178.967,6.207,149.426
C04465=1130.684,-60.798,-47.068,178.969,6.208,149.426
C04466=1130.679,-60.548,-47.079,178.971,6.209,149.425
C04467=1130.674,-60.298,-47.090,178.973,6.209,149.425
C04468=1130.669,-60.048,-47.100,178.975,6.209,149.424
C04469=1130.663,-59.799,-47.110,178.978,6.210,149.423
C04470=1130.657,-59.549,-47.121,178.980,6.211,149.423
C04471=1130.652,-59.299,-47.131,178.982,6.211,149.422
C04472=1130.647,-59.050,-47.142,178.984,6.212,149.422
C04473=1130.642,-58.800,-47.153,178.987,6.213,149.421
C04474=1130.637,-58.550,-47.163,178.989,6.213,149.421
C04475=1130.632,-58.300,-47.173,178.991,6.213,149.420
C04476=1130.626,-58.051,-47.184,178.993,6.214,149.420
C04477=1130.621,-57.801,-47.195,178.996,6.214,149.419
C04478=1130.616,-57.551,-47.205,178.998,6.215,149.419
C04479=1130.611,-57.301,-47.216,179.000,6.216,149.418
C04480=1130.605,-57.052,-47.227,179.002,6.217,149.418
C04481=1130.600,-56.802,-47.237,179.004,6.218,149.417
C04482=1130.595,-56.552,-47.247,179.007,6.218,149.416
C04483=1130.589,-56.303,-47.258,179.009,6.219,149.416
C04484=1130.585,-56.053,-47.269,179.011,6.219,149.416
C04485=1130.579,-55.804,-47.279,179.013,6.219,149.415
C04486=1130.574,-55.554,-47.290,179.015,6.220,149.415
C04487=1130.569,-55.304,-47.301,179.018,6.221,149.414
C04488=1130.563,-55.054,-47.312,179.020,6.221,149.413
C04489=1130.558,-54.805,-47.323,179.022,6.222,149.413
C04490=1130.553,-54.555,-47.333,179.024,6.223,149.412
C04491=1130.547,-54.305,-47.344,179.027,6.224,149.412
C04492=1130.542,-54.055,-47.355,179.029,6.224,149.411
C04493=1130.537,-53.806,-47.365,179.031,6.225,149.411
C04494=1130.532,-53.556,-47.376,179.034,6.226,149.410
C04495=1130.526,-53.307,-47.387,179.035,6.226,149.410
C04496=1130.521,-53.056,-47.398,179.038,6.226,149.409
C04497=1130.515,-52.807,-47.409,179.040,6.227,149.409
C04498=1130.510,-52.557,-47.419,179.042,6.227,149.408
C04499=1130.505,-52.307,-47.430,179.044,6.228,149.408
C04500=1130.500,-52.058,-47.441,179.047,6.229,149.407
C04501=1130.495,-51.808,-47.451,179.049,6.229,149.406
C04502=1130.489,-51.558,-47.463,179.052,6.230,149.406
C04503=1130.484,-51.287,-47.474,179.054,6.231,149.406
C04504=1130.478,-51.017,-47.486,179.056,6.231,149.405
C04505=1130.472,-50.746,-47.498,179.059,6.232,149.404
C04506=1130.466,-50.475,-47.510,179.061,6.232,149.404
C04507=1130.461,-50.225,-47.520,179.063,6.233,149.403
C04508=1130.456,-49.976,-47.532,179.066,6.234,149.403
C04509=1130.451,-49.726,-47.542,179.068,6.235,149.402
C04510=1130.446,-49.477,-47.553,179.070,6.235,149.402
C04511=1130.440,-49.226,-47.564,179.073,6.236,149.401
C04512=1130.435,-48.977,-47.575,179.075,6.237,149.401
C04513=1130.430,-48.727,-47.586,179.077,6.237,149.400
C04514=1130.425,-48.478,-47.597,179.079,6.238,149.400
C04515=1130.419,-48.227,-47.608,179.082,6.239,149.399
C04516=1130.414,-47.978,-47.619,179.084,6.239,149.398
C04517=1130.409,-47.728,-47.629,179.086,6.240,149.398
C04518=1130.403,-47.478,-47.641,179.089,6.241,149.397
C04519=1130.397,-47.229,-47.651,179.091,6.240,149.397
C04520=1130.393,-46.979,-47.663,179.093,6.241,149.396
C04521=1130.387,-46.730,-47.674,179.095,6.242,149.396
C04522=1130.382,-46.480,-47.685,179.097,6.243,149.395
C04523=1130.377,-46.230,-47.696,179.100,6.243,149.395
C04524=1130.371,-45.980,-47.706,179.102,6.244,149.394
C04525=1130.366,-45.730,-47.718,179.104,6.245,149.394
C04526=1130.361,-45.481,-47.730,179.106,6.245,149.393
C04527=1130.356,-45.231,-47.740,179.109,6.246,149.393
C04528=1130.350,-44.981,-47.752,179.111,6.247,149.392
C04529=1130.345,-44.731,-47.762,179.113,6.247,149.391
C04530=1130.340,-44.482,-47.773,179.116,6.248,149.391
C04531=1130.335,-44.232,-47.785,179.118,6.249,149.391
C04532=1130.329,-43.983,-47.795,179.120,6.249,149.390
C04533=1130.324,-43.733,-47.807,179.123,6.250,149.389
C04534=1130.319,-43.483,-47.818,179.125,6.251,149.389
C04535=1130.314,-43.234,-47.829,179.127,6.252,149.388
C04536=1130.309,-42.984,-47.840,179.130,6.252,149.388
C04537=1130.303,-42.734,-47.852,179.132,6.253,149.387
C04538=1130.298,-42.485,-47.863,179.134,6.254,149.387
C04539=1130.292,-42.235,-47.874,179.136,6.254,149.386
C04540=1130.287,-41.985,-47.885,179.139,6.255,149.386
C04541=1130.283,-41.735,-47.896,179.141,6.256,149.385
C04542=1130.277,-41.486,-47.908,179.143,6.256,149.385
C04543=1130.272,-41.236,-47.919,179.146,6.257,149.384
C04544=1130.266,-40.986,-47.930,179.148,6.257,149.383
C04545=1130.261,-40.737,-47.941,179.150,6.258,149.383
C04546=1130.256,-40.487,-47.953,179.153,6.259,149.382
C04547=1130.251,-40.237,-47.964,179.155,6.260,149.382
C04548=1130.245,-39.988,-47.975,179.157,6.260,149.381
C04549=1130.240,-39.738,-47.987,179.160,6.261,149.381
C04550=1130.235,-39.488,-47.998,179.162,6.262,149.380
C04551=1130.230,-39.238,-48.010,179.164,6.262,149.380
C04552=1130.224,-38.989,-48.021,179.167,6.263,149.379
C04553=1130.219,-38.739,-48.032,179.169,6.264,149.379
C04554=1130.214,-38.489,-48.043,179.171,6.264,149.378
C04555=1130.209,-38.239,-48.055,179.173,6.265,149.378
C04556=1130.203,-37.990,-48.066,179.176,6.266,149.377
C04557=1130.198,-37.740,-48.078,179.178,6.266,149.377
C04558=1130.193,-37.491,-48.089,179.180,6.267,149.376
C04559=1130.187,-37.241,-48.100,179.182,6.268,149.376
C04560=1130.182,-36.991,-48.111,179.185,6.268,149.375
C04561=1130.177,-36.741,-48.123,179.187,6.269,149.374
C04562=1130.172,-36.492,-48.134,179.189,6.270,149.374
C04563=1130.167,-36.242,-48.146,179.192,6.270,149.373
C04564=1130.161,-35.993,-48.157,179.194,6.271,149.373
C04565=1130.156,-35.743,-48.169,179.197,6.272,149.372
C04566=1130.151,-35.493,-48.180,179.199,6.273,149.372
C04567=1130.146,-35.243,-48.192,179.201,6.273,149.371
C04568=1130.140,-34.995,-48.203,179.204,6.274,149.371
C04569=1130.135,-34.745,-48.215,179.206,6.275,149.370
C04570=1130.130,-34.495,-48.226,179.208,6.275,149.370
C04571=1130.125,-34.245,-48.238,179.211,6.276,149.369
C04572=1130.119,-33.995,-48.250,179.213,6.276,149.369
C04573=1130.114,-33.746,-48.261,179.215,6.277,149.368
C04574=1130.109,-33.496,-48.273,179.217,6.278,149.368
C04575=1130.104,-33.247,-48.284,179.220,6.278,149.367
C04576=1130.099,-32.997,-48.296,179.222,6.279,149.366
C04577=1130.093,-32.747,-48.308,179.224,6.280,149.366
C04578=1130.089,-32.497,-48.319,179.226,6.281,149.365
C04579=1130.082,-32.248,-48.331,179.229,6.281,149.365
C04580=1130.078,-31.998,-48.342,179.231,6.282,149.364
C04581=1130.072,-31.748,-48.354,179.233,6.283,149.364
C04582=1130.067,-31.498,-48.366,179.236,6.283,149.363
C04583=1130.062,-31.249,-48.377,179.239,6.285,149.363
C04584=1130.057,-30.999,-48.389,179.241,6.285,149.362
C04585=1130.051,-30.750,-48.401,179.243,6.286,149.362
C04586=1130.046,-30.500,-48.412,179.246,6.287,149.361
C04587=1130.041,-30.250,-48.424,179.248,6.287,149.361
C04588=1130.035,-30.000,-48.436,179.250,6.288,149.360
C04589=1130.031,-29.751,-48.448,179.252,6.289,149.360
C04590=1130.025,-29.501,-48.460,179.255,6.289,149.359
C04591=1130.020,-29.251,-48.471,179.257,6.290,149.358
C04592=1130.015,-29.002,-48.483,179.260,6.291,149.358
C04593=1130.009,-28.752,-48.494,179.262,6.291,149.357
C04594=1130.004,-28.502,-48.506,179.264,6.292,149.357
C04595=1129.999,-28.253,-48.518,179.267,6.293,149.356
C04596=1129.994,-28.003,-48.530,179.269,6.294,149.356
C04597=1129.989,-27.753,-48.542,179.271,6.294,149.355
C04598=1129.984,-27.504,-48.553,179.274,6.295,149.355
C04599=1129.978,-27.254,-48.565,179.276,6.296,149.354
C04600=1129.973,-27.004,-48.577,179.279,6.297,149.354
C04601=1129.968,-26.755,-48.590,179.281,6.298,149.353
C04602=1129.963,-26.505,-48.601,179.283,6.298,149.352
C04603=1129.958,-26.255,-48.613,179.286,6.299,149.352
C04604=1129.952,-26.005,-48.625,179.288,6.300,149.351
C04605=1129.947,-25.757,-48.637,179.290,6.300,149.351
C04606=1129.942,-25.507,-48.648,179.293,6.301,149.350
C04607=1129.936,-25.236,-48.662,179.295,6.301,149.350
C04608=1129.931,-24.966,-48.675,179.298,6.303,149.349
C04609=1129.925,-24.696,-48.687,179.300,6.304,149.349
C04610=1129.919,-24.426,-48.700,179.303,6.304,149.348
C04611=1129.914,-24.176,-48.712,179.305,6.305,149.348
C04612=1129.909,-23.927,-48.725,179.308,6.305,149.347
C04613=1129.904,-23.677,-48.736,179.310,6.306,149.346
C04614=1129.899,-23.427,-48.748,179.313,6.308,149.346
C04615=1129.894,-23.178,-48.761,179.315,6.309,149.345
C04616=1129.888,-22.928,-48.772,179.318,6.309,149.345
C04617=1129.883,-22.678,-48.784,179.320,6.310,149.344
C04618=1129.878,-22.429,-48.797,179.322,6.311,149.344
C04619=1129.873,-22.179,-48.808,179.324,6.311,149.343
C04620=1129.867,-21.929,-48.820,179.327,6.312,149.343
C04621=1129.862,-21.680,-48.833,179.329,6.312,149.342
C04622=1129.857,-21.430,-48.845,179.331,6.313,149.342
C04623=1129.851,-21.180,-48.856,179.334,6.314,149.341
C04624=1129.846,-20.931,-48.869,179.337,6.315,149.341
C04625=1129.841,-20.681,-48.881,179.339,6.316,149.340
C04626=1129.836,-20.431,-48.894,179.341,6.317,149.340
C04627=1129.831,-20.182,-48.905,179.344,6.317,149.339
C04628=1129.826,-19.932,-48.917,179.346,6.318,149.338
C04629=1129.821,-19.682,-48.929,179.348,6.319,149.338
C04630=1129.815,-19.432,-48.941,179.351,6.319,149.337
C04631=1129.810,-19.183,-48.954,179.353,6.321,149.337
C04632=1129.805,-18.933,-48.966,179.356,6.322,149.336
C04633=1129.799,-18.684,-48.978,179.358,6.322,149.336
C04634=1129.794,-18.434,-48.990,179.361,6.323,149.335
C04635=1129.789,-18.185,-49.003,179.363,6.324,149.335
C04636=1129.783,-17.935,-49.015,179.365,6.324,149.334
C04637=1129.778,-17.685,-49.027,179.368,6.325,149.333
C04638=1129.773,-17.435,-49.039,179.370,6.326,149.333
C04639=1129.768,-17.186,-49.052,179.373,6.327,149.333
C04640=1129.763,-16.937,-49.064,179.375,6.328,149.332
C04641=1129.757,-16.687,-49.076,179.377,6.328,149.331
C04642=1129.752,-16.438,-49.089,179.380,6.329,149.331
C04643=1129.747,-16.187,-49.101,179.382,6.330,149.330
C04644=1129.742,-15.938,-49.114,179.384,6.330,149.330
C04645=1129.737,-15.688,-49.126,179.387,6.332,149.329
C04646=1129.732,-15.438,-49.138,179.389,6.333,149.329
C04647=1129.726,-15.189,-49.151,179.392,6.333,149.328
C04648=1129.721,-14.939,-49.163,179.394,6.334,149.328
C04649=1129.716,-14.690,-49.175,179.396,6.335,149.327
C04650=1129.710,-14.440,-49.187,179.399,6.335,149.327
C04651=1129.705,-14.191,-49.200,179.401,6.336,149.326
C04652=1129.701,-13.940,-49.213,179.404,6.337,149.326
C04653=1129.695,-13.691,-49.225,179.406,6.338,149.325
C04654=1129.690,-13.441,-49.237,179.409,6.339,149.324
C04655=1129.685,-13.192,-49.250,179.411,6.339,149.324
C04656=1129.680,-12.942,-49.262,179.413,6.340,149.323
C04657=1129.675,-12.693,-49.274,179.415,6.341,149.323
C04658=1129.669,-12.443,-49.287,179.419,6.342,149.322
C04659=1129.665,-12.193,-49.299,179.421,6.343,149.322
C04660=1129.660,-11.943,-49.312,179.423,6.344,149.321
C04661=1129.654,-11.694,-49.324,179.426,6.344,149.321
C04662=1129.649,-11.445,-49.337,179.428,6.345,149.320
C04663=1129.643,-11.194,-49.349,179.431,6.346,149.320
C04664=1129.638,-10.945,-49.362,179.433,6.347,149.319
C04665=1129.633,-10.695,-49.375,179.435,6.348,149.319
C04666=1129.628,-10.446,-49.388,179.438,6.348,149.318
C04667=1129.623,-10.196,-49.399,179.440,6.349,149.318
C04668=1129.618,-9.947,-49.412,179.443,6.350,149.317
C04669=1129.613,-9.697,-49.425,179.445,6.351,149.316
C04670=1129.608,-9.448,-49.437,179.447,6.352,149.316
C04671=1129.602,-9.198,-49.451,179.450,6.352,149.315
C04672=1129.597,-8.948,-49.463,179.452,6.353,149.315
C04673=1129.592,-8.698,-49.475,179.455,6.354,149.314
C04674=1129.587,-8.449,-49.488,179.457,6.356,149.314
C04675=1129.582,-8.199,-49.501,179.460,6.356,149.313
C04676=1129.577,-7.950,-49.513,179.462,6.357,149.313
C04677=1129.571,-7.700,-49.527,179.464,6.358,149.312
C04678=1129.566,-7.450,-49.539,179.468,6.359,149.312
C04679=1129.561,-7.201,-49.551,179.470,6.360,149.311
C04680=1129.556,-6.951,-49.564,179.472,6.360,149.311
C04681=1129.551,-6.702,-49.577,179.474,6.361,149.310
C04682=1129.545,-6.452,-49.590,179.477,6.362,149.309
C04683=1129.540,-6.203,-49.603,179.480,6.363,149.309
C04684=1129.535,-5.953,-49.615,179.482,6.364,149.309
C04685=1129.530,-5.703,-49.628,179.484,6.364,149.308
C04686=1129.524,-5.454,-49.641,179.487,6.365,149.307
C04687=1129.519,-5.204,-49.654,179.489,6.366,149.307
C04688=1129.514,-4.954,-49.666,179.492,6.367,149.306
C04689=1129.509,-4.704,-49.679,179.494,6.368,149.306
C04690=1129.503,-4.455,-49.692,179.496,6.369,149.305
C04691=1129.499,-4.205,-49.705,179.499,6.370,149.305
C04692=1129.494,-3.955,-49.717,179.502,6.371,149.304
C04693=1129.489,-3.706,-49.730,179.504,6.372,149.304
C04694=1129.483,-3.456,-49.743,179.506,6.372,149.303
C04695=1129.478,-3.206,-49.756,179.509,6.373,149.302
C04696=1129.473,-2.957,-49.769,179.512,6.374,149.302
C04697=1129.467,-2.707,-49.782,179.514,6.375,149.302
C04698=1129.463,-2.457,-49.795,179.516,6.376,149.301
C04699=1129.458,-2.208,-49.808,179.519,6.376,149.300
C04700=1129.452,-1.959,-49.822,179.521,6.378,149.300
C04701=1129.448,-1.709,-49.834,179.524,6.379,149.299
C04702=1129.442,-1.460,-49.847,179.526,6.379,149.299
C04703=1129.437,-1.210,-49.860,179.528,6.380,149.298
C04704=1129.432,-0.960,-49.873,179.531,6.382,149.298
C04705=1129.427,-0.711,-49.886,179.534,6.382,149.297
C04706=1129.421,-0.461,-49.899,179.536,6.383,149.297
C04707=1129.417,-0.211,-49.912,179.538,6.384,149.296
C04708=1129.411,0.038,-49.925,179.541,6.385,149.296
C04709=1129.406,0.288,-49.938,179.544,6.386,149.295
C04710=1129.401,0.537,-49.951,179.546,6.386,149.295
C04711=1129.395,0.807,-49.965,179.549,6.388,149.294
C04712=1129.369,2.067,-50.034,179.580,6.350,149.277
C04713=1129.364,2.318,-50.048,179.580,6.354,149.277
C04714=1129.359,2.567,-50.060,179.581,6.359,149.278
C04715=1129.355,2.816,-50.074,179.582,6.363,149.279
C04716=1129.349,3.066,-50.087,179.582,6.368,149.280
C04717=1129.344,3.315,-50.100,179.583,6.373,149.281
C04718=1129.338,3.566,-50.113,179.583,6.377,149.282
C04719=1129.334,3.814,-50.127,179.583,6.382,149.283
C04720=1129.328,4.065,-50.140,179.584,6.386,149.283
C04721=1129.323,4.314,-50.153,179.585,6.391,149.284
C04722=1129.318,4.564,-50.166,179.585,6.395,149.285
C04723=1129.313,4.813,-50.180,179.585,6.399,149.286
C04724=1129.307,5.063,-50.193,179.586,6.404,149.287
C04725=1129.303,5.313,-50.206,179.586,6.409,149.288
C04726=1129.297,5.562,-50.219,179.586,6.413,149.288
C04727=1129.293,5.812,-50.233,179.587,6.417,149.289
C04728=1129.287,6.061,-50.246,179.587,6.422,149.290
C04729=1129.282,6.311,-50.259,179.588,6.427,149.291
C04730=1129.277,6.560,-50.273,179.588,6.431,149.292
C04731=1129.272,6.810,-50.285,179.589,6.435,149.293
C04732=1129.265,7.154,-50.304,179.589,6.441,149.294
C04733=1129.257,7.498,-50.322,179.590,6.447,149.295
C04734=1129.250,7.843,-50.341,179.590,6.454,149.296
C04735=1129.243,8.187,-50.359,179.591,6.459,149.297
C04736=1129.239,8.436,-50.373,179.592,6.465,149.298
C04737=1129.233,8.686,-50.386,179.592,6.470,149.299
C04738=1129.228,8.935,-50.400,179.593,6.474,149.300
C04739=1129.223,9.185,-50.413,179.595,6.479,149.301
C04740=1129.218,9.434,-50.427,179.596,6.484,149.301
C04741=1129.213,9.684,-50.440,179.596,6.489,149.302
C04742=1129.207,9.934,-50.453,179.597,6.493,149.303
C04743=1129.202,10.183,-50.467,179.598,6.498,149.304
C04744=1129.197,10.433,-50.480,179.599,6.503,149.305
C04745=1129.192,10.682,-50.494,179.600,6.507,149.305
C04746=1129.186,10.932,-50.508,179.600,6.512,149.306
C04747=1129.182,11.181,-50.521,179.602,6.517,149.307
C04748=1129.177,11.431,-50.535,179.603,6.522,149.308
C04749=1129.171,11.681,-50.549,179.604,6.526,149.308
C04750=1129.167,11.930,-50.562,179.604,6.531,149.309
C04751=1129.161,12.180,-50.576,179.606,6.536,149.310
C04752=1129.156,12.429,-50.590,179.606,6.541,149.311
C04753=1129.151,12.679,-50.603,179.607,6.545,149.311
C04754=1129.146,12.928,-50.617,179.608,6.550,149.312
C04755=1129.141,13.178,-50.631,179.610,6.555,149.313
C04756=1129.135,13.428,-50.644,179.611,6.559,149.314
C04757=1129.131,13.677,-50.658,179.611,6.564,149.314
C04758=1129.125,13.927,-50.671,179.612,6.568,149.315
C04759=1129.120,14.176,-50.685,179.613,6.573,149.316
C04760=1129.115,14.426,-50.699,179.614,6.578,149.317
C04761=1129.110,14.676,-50.712,179.616,6.583,149.317
C04762=1129.105,14.925,-50.726,179.616,6.587,149.318
C04763=1129.100,15.175,-50.741,179.617,6.592,149.319
C04764=1129.094,15.424,-50.755,179.618,6.597,149.320
C04765=1129.090,15.674,-50.768,179.619,6.601,149.320
C04766=1129.085,15.924,-50.782,179.620,6.606,149.321
C04767=1129.079,16.173,-50.796,179.621,6.610,149.322
C04768=1129.074,16.423,-50.809,179.622,6.615,149.322
C04769=1129.069,16.673,-50.824,179.624,6.620,149.323
C04770=1129.063,16.922,-50.837,179.624,6.625,149.324
C04771=1129.059,17.171,-50.851,179.625,6.629,149.325
C04772=1129.054,17.421,-50.865,179.626,6.633,149.325
C04773=1129.048,17.670,-50.879,179.627,6.638,149.326
C04774=1129.043,17.920,-50.893,179.628,6.642,149.327
C04775=1129.039,18.170,-50.907,179.630,6.647,149.327
C04776=1129.033,18.419,-50.921,179.631,6.652,149.328
C04777=1129.028,18.668,-50.935,179.631,6.656,149.329
C04778=1129.024,18.918,-50.949,179.632,6.661,149.330
C04779=1129.018,19.167,-50.962,179.633,6.665,149.330
C04780=1129.013,19.417,-50.976,179.634,6.671,149.331
C04781=1129.008,19.667,-50.991,179.635,6.675,149.332
C04782=1129.003,19.917,-51.005,179.636,6.679,149.332
C04783=1128.998,20.166,-51.019,179.637,6.684,149.333
C04784=1128.993,20.381,-51.031,179.639,6.688,149.334
C04785=1128.988,20.596,-51.043,179.639,6.691,149.334
C04786=1128.985,20.812,-51.056,179.640,6.696,149.335
C04787=1128.980,21.027,-51.068,179.641,6.699,149.335
C04788=1128.976,21.243,-51.080,179.642,6.703,149.336
C04789=1128.971,21.458,-51.092,179.643,6.708,149.337
C04790=1128.967,21.673,-51.104,179.643,6.711,149.337
C04791=1128.962,21.888,-51.117,179.645,6.715,149.338
C04792=1128.957,22.138,-51.131,179.646,6.719,149.338
C04793=1128.952,22.388,-51.145,179.647,6.724,149.339
C04794=1128.947,22.637,-51.159,179.648,6.728,149.340
C04795=1128.942,22.887,-51.173,179.649,6.733,149.341
C04796=1128.937,23.136,-51.188,179.650,6.738,149.341
C04797=1128.932,23.386,-51.202,179.651,6.742,149.342
C04798=1128.927,23.636,-51.216,179.652,6.746,149.343
C04799=1128.922,23.885,-51.230,179.653,6.751,149.343
C04800=1128.917,24.134,-51.244,179.654,6.755,149.344
C04801=1128.912,24.384,-51.259,179.655,6.760,149.345
C04802=1128.907,24.634,-51.273,179.656,6.764,149.345
C04803=1128.902,24.883,-51.288,179.657,6.768,149.346
C04804=1128.896,25.132,-51.302,179.659,6.773,149.347
C04805=1128.891,25.382,-51.317,179.660,6.778,149.347
C04806=1128.886,25.632,-51.331,179.661,6.782,149.348
C04807=1128.881,25.881,-51.345,179.662,6.786,149.349
C04808=1128.876,26.131,-51.360,179.663,6.791,149.349
C04809=1128.871,26.381,-51.374,179.664,6.795,149.350
C04810=1128.866,26.630,-51.389,179.665,6.799,149.351
C04811=1128.861,26.879,-51.403,179.666,6.804,149.351
C04812=1128.856,27.129,-51.417,179.668,6.809,149.352
C04813=1128.850,27.379,-51.432,179.669,6.813,149.353
C04814=1128.845,27.628,-51.447,179.670,6.817,149.353
C04815=1128.841,27.877,-51.461,179.671,6.822,149.354
C04816=1128.836,28.127,-51.475,179.672,6.826,149.354
C04817=1128.831,28.377,-51.490,179.673,6.830,149.355
C04818=1128.826,28.626,-51.505,179.674,6.835,149.356
C04819=1128.820,28.875,-51.519,179.675,6.839,149.356
C04820=1128.815,29.125,-51.533,179.676,6.843,149.357
C04821=1128.810,29.375,-51.548,179.678,6.848,149.358
C04822=1128.805,29.624,-51.563,179.679,6.853,149.358
C04823=1128.800,29.874,-51.577,179.680,6.857,149.359
C04824=1128.794,30.124,-51.592,179.681,6.861,149.360
C04825=1128.790,30.373,-51.607,179.682,6.866,149.360
C04826=1128.785,30.622,-51.621,179.683,6.870,149.361
C04827=1128.780,30.871,-51.636,179.684,6.874,149.362
C04828=1128.775,31.121,-51.651,179.685,6.879,149.362
C04829=1128.770,31.371,-51.665,179.686,6.883,149.363
C04830=1128.765,31.620,-51.680,179.688,6.887,149.364
C04831=1128.760,31.870,-51.695,179.689,6.892,149.364
C04832=1128.755,32.119,-51.710,179.690,6.897,149.365
C04833=1128.750,32.369,-51.724,179.692,6.901,149.365
C04834=1128.745,32.619,-51.739,179.693,6.905,149.366
C04835=1128.739,32.868,-51.754,179.694,6.909,149.367
C04836=1128.734,33.118,-51.769,179.695,6.914,149.367
C04837=1128.730,33.367,-51.784,179.696,6.918,149.368
C04838=1128.723,33.616,-51.798,179.697,6.922,149.368
C04839=1128.719,33.865,-51.813,179.698,6.927,149.369
C04840=1128.715,34.081,-51.826,179.700,6.930,149.370
C04841=1128.710,34.297,-51.839,179.700,6.934,149.370
C04842=1128.706,34.511,-51.851,179.702,6.938,149.371
C04843=1128.702,34.727,-51.864,179.703,6.941,149.371
C04844=1128.697,34.942,-51.877,179.704,6.945,149.372
C04845=1128.693,35.157,-51.890,179.705,6.948,149.372
C04846=1128.688,35.373,-51.903,179.706,6.953,149.373
C04847=1128.684,35.588,-51.916,179.707,6.956,149.373
C04848=1128.679,35.837,-51.931,179.708,6.960,149.374
C04849=1128.674,36.087,-51.945,179.709,6.965,149.375
C04850=1128.669,36.336,-51.961,179.710,6.969,149.375
C04851=1128.664,36.585,-51.976,179.711,6.973,149.376
C04852=1128.658,36.835,-51.991,179.712,6.977,149.376
C04853=1128.654,37.085,-52.006,179.713,6.981,149.377
C04854=1128.648,37.335,-52.021,179.715,6.986,149.378
C04855=1128.644,37.584,-52.036,179.717,6.990,149.378
C04856=1128.638,37.833,-52.051,179.718,6.995,149.379
C04857=1128.633,38.083,-52.066,179.719,6.999,149.379
C04858=1128.628,38.333,-52.081,179.720,7.003,149.380
C04859=1128.624,38.582,-52.096,179.721,7.007,149.380
C04860=1128.618,38.831,-52.112,179.723,7.012,149.381
C04861=1128.613,39.081,-52.126,179.724,7.016,149.382
C04862=1128.608,39.330,-52.142,179.725,7.020,149.382
C04863=1128.603,39.580,-52.157,179.726,7.024,149.383
C04864=1128.598,39.829,-52.172,179.727,7.028,149.383
C04865=1128.593,40.079,-52.187,179.728,7.033,149.384
C04866=1128.588,40.328,-52.202,179.729,7.037,149.385
C04867=1128.584,40.578,-52.218,179.731,7.041,149.385
C04868=1128.578,40.827,-52.233,179.732,7.045,149.386
C04869=1128.573,41.077,-52.248,179.733,7.050,149.386
C04870=1128.568,41.326,-52.263,179.735,7.054,149.387
C04871=1128.563,41.575,-52.278,179.736,7.058,149.387
C04872=1128.558,41.825,-52.294,179.737,7.062,149.388
C04873=1128.552,42.074,-52.309,179.738,7.066,149.388
C04874=1128.548,42.324,-52.325,179.739,7.070,149.389
C04875=1128.543,42.573,-52.340,179.740,7.075,149.390
C04876=1128.538,42.823,-52.355,179.742,7.079,149.390
C04877=1128.533,43.073,-52.370,179.743,7.083,149.391
C04878=1128.527,43.322,-52.386,179.744,7.087,149.391
C04879=1128.523,43.572,-52.401,179.746,7.091,149.392
C04880=1128.518,43.821,-52.417,179.747,7.095,149.393
C04881=1128.512,44.071,-52.432,179.748,7.100,149.393
C04882=1128.508,44.320,-52.447,179.749,7.104,149.394
C04883=1128.502,44.569,-52.463,179.751,7.108,149.394
C04884=1128.498,44.819,-52.479,179.752,7.112,149.395
C04885=1128.493,45.068,-52.494,179.753,7.116,149.395
C04886=1128.488,45.318,-52.509,179.754,7.120,149.396
C04887=1128.482,45.567,-52.525,179.756,7.124,149.396
C04888=1128.478,45.817,-52.540,179.757,7.129,149.397
C04889=1128.473,46.066,-52.556,179.758,7.133,149.397
C04890=1128.467,46.316,-52.572,179.760,7.138,149.398
C04891=1128.462,46.565,-52.587,179.761,7.142,149.399
C04892=1128.458,46.815,-52.602,179.763,7.146,149.399
C04893=1128.453,47.064,-52.618,179.764,7.150,149.400
C04894=1128.447,47.314,-52.634,179.765,7.154,149.400
C04895=1128.443,47.563,-52.649,179.766,7.158,149.401
C04896=1128.438,47.778,-52.663,179.767,7.162,149.401
C04897=1128.433,47.993,-52.676,179.768,7.165,149.402
C04898=1128.429,48.209,-52.690,179.770,7.169,149.402
C04899=1128.425,48.423,-52.703,179.770,7.172,149.403
C04900=1128.421,48.639,-52.717,179.772,7.176,149.403
C04901=1128.417,48.854,-52.730,179.773,7.179,149.404
C04902=1128.412,49.069,-52.744,179.774,7.183,149.404
C04903=1128.408,49.285,-52.758,179.775,7.186,149.405
C04904=1128.403,49.534,-52.773,179.776,7.191,149.405
C04905=1128.398,49.783,-52.788,179.778,7.194,149.406
C04906=1128.393,50.032,-52.805,179.779,7.199,149.406
C04907=1128.388,50.282,-52.821,179.781,7.203,149.407
C04908=1128.383,50.531,-52.836,179.782,7.207,149.407
C04909=1128.378,50.782,-52.852,179.783,7.211,149.408
C04910=1128.374,51.030,-52.868,179.784,7.215,149.408
C04911=1128.368,51.279,-52.883,179.785,7.220,149.409
C04912=1128.364,51.530,-52.899,179.787,7.223,149.409
C04913=1128.358,51.779,-52.915,179.788,7.228,149.410
C04914=1128.353,52.028,-52.931,179.790,7.232,149.411
C04915=1128.348,52.278,-52.947,179.791,7.236,149.411
C04916=1128.343,52.527,-52.963,179.792,7.240,149.412
C04917=1128.338,52.776,-52.979,179.794,7.244,149.412
C04918=1128.333,53.026,-52.995,179.795,7.248,149.413
C04919=1128.328,53.276,-53.011,179.796,7.252,149.413
C04920=1128.323,53.525,-53.027,179.798,7.256,149.414
C04921=1128.319,53.774,-53.042,179.799,7.260,149.414
C04922=1128.313,54.024,-53.058,179.800,7.264,149.415
C04923=1128.309,54.273,-53.075,179.802,7.268,149.415
C04924=1128.303,54.522,-53.090,179.803,7.273,149.416
C04925=1128.299,54.772,-53.107,179.804,7.277,149.416
C04926=1128.293,55.021,-53.122,179.805,7.281,149.417
C04927=1128.288,55.271,-53.138,179.807,7.285,149.417
C04928=1128.284,55.520,-53.155,179.809,7.289,149.418
C04929=1128.278,55.770,-53.170,179.810,7.293,149.418
C04930=1128.274,56.019,-53.187,179.811,7.297,149.419
C04931=1128.268,56.268,-53.203,179.812,7.301,149.420
C04932=1128.264,56.518,-53.219,179.814,7.305,149.420
C04933=1128.258,56.767,-53.235,179.815,7.309,149.421
C04934=1128.254,57.017,-53.251,179.817,7.313,149.421
C04935=1128.249,57.266,-53.267,179.818,7.317,149.421
C04936=1128.243,57.516,-53.284,179.819,7.322,149.422
C04937=1128.238,57.765,-53.300,179.821,7.325,149.422
C04938=1128.233,58.015,-53.317,179.822,7.330,149.423
C04939=1128.228,58.264,-53.332,179.823,7.334,149.424
C04940=1128.223,58.513,-53.348,179.825,7.338,149.424
C04941=1128.219,58.763,-53.365,179.826,7.342,149.425
C04942=1128.213,59.012,-53.381,179.828,7.346,149.425
C04943=1128.209,59.261,-53.397,179.829,7.350,149.425
C04944=1128.204,59.512,-53.413,179.830,7.354,149.426
C04945=1128.199,59.760,-53.430,179.832,7.358,149.427
C04946=1128.194,60.010,-53.446,179.833,7.362,149.427
C04947=1128.188,60.260,-53.462,179.835,7.366,149.428
C04948=1128.184,60.509,-53.479,179.835,7.369,149.428
C04949=1128.179,60.758,-53.495,179.837,7.374,149.429
C04950=1128.174,61.008,-53.511,179.838,7.377,149.429
C04951=1128.169,61.257,-53.528,179.840,7.381,149.430
C04952=1128.164,61.472,-53.542,179.841,7.385,149.430
C04953=1128.161,61.687,-53.556,179.842,7.388,149.430
C04954=1128.156,61.902,-53.571,179.843,7.393,149.431
C04955=1128.152,62.117,-53.584,179.844,7.396,149.431
C04956=1128.147,62.333,-53.599,179.846,7.400,149.432
C04957=1128.143,62.547,-53.612,179.847,7.403,149.432
C04958=1128.138,62.762,-53.627,179.848,7.406,149.433
C04959=1128.135,62.977,-53.641,179.849,7.410,149.433
C04960=1128.130,63.227,-53.658,179.851,7.414,149.434
C04961=1128.124,63.476,-53.675,179.852,7.418,149.434
C04962=1128.120,63.726,-53.691,179.854,7.422,149.435
C04963=1128.115,63.975,-53.707,179.855,7.426,149.435
C04964=1128.110,64.224,-53.724,179.857,7.430,149.436
C04965=1128.105,64.474,-53.741,179.858,7.434,149.436
C04966=1128.100,64.723,-53.757,179.859,7.438,149.437
C04967=1128.095,64.973,-53.773,179.861,7.442,149.437
C04968=1128.090,65.222,-53.790,179.862,7.446,149.438
C04969=1128.085,65.472,-53.807,179.864,7.450,149.438
C04970=1128.080,65.721,-53.823,179.865,7.454,149.439
C04971=1128.075,65.970,-53.840,179.866,7.457,149.439
C04972=1128.070,66.220,-53.857,179.867,7.461,149.440
C04973=1128.065,66.469,-53.874,179.869,7.465,149.440
C04974=1128.060,66.718,-53.890,179.870,7.469,149.440
C04975=1128.055,66.968,-53.907,179.871,7.474,149.441
C04976=1128.051,67.217,-53.924,179.873,7.477,149.442
C04977=1128.046,67.466,-53.940,179.875,7.481,149.442
C04978=1128.040,67.716,-53.958,179.876,7.486,149.443
C04979=1128.036,67.965,-53.974,179.877,7.490,149.443
C04980=1128.031,68.214,-53.990,179.879,7.493,149.443
C04981=1128.026,68.464,-54.008,179.880,7.497,149.444
C04982=1128.021,68.713,-54.024,179.882,7.502,149.445
C04983=1128.016,68.963,-54.042,179.883,7.506,149.445
C04984=1128.011,69.212,-54.058,179.885,7.509,149.445
C04985=1128.006,69.461,-54.075,179.886,7.513,149.446
C04986=1128.001,69.711,-54.092,179.887,7.518,149.446
C04987=1127.996,69.960,-54.108,179.889,7.522,149.447
C04988=1127.991,70.210,-54.125,179.891,7.525,149.447
C04989=1127.986,70.459,-54.142,179.892,7.530,149.448
C04990=1127.981,70.709,-54.159,179.893,7.534,149.448
C04991=1127.976,70.958,-54.176,179.895,7.538,149.449
C04992=1127.972,71.207,-54.192,179.896,7.541,149.449
C04993=1127.967,71.457,-54.210,179.898,7.546,149.450
C04994=1127.962,71.706,-54.227,179.899,7.550,149.450
C04995=1127.956,71.955,-54.244,179.901,7.554,149.451
C04996=1127.952,72.205,-54.261,179.902,7.557,149.451
C04997=1127.947,72.454,-54.278,179.903,7.562,149.452
C04998=1127.942,72.704,-54.295,179.905,7.566,149.452
C04999=1127.937,72.953,-54.313,179.907,7.570,149.453
C05000=1127.932,73.202,-54.329,179.908,7.573,149.453
C05001=1127.927,73.452,-54.346,179.909,7.578,149.454
C05002=1127.922,73.701,-54.363,179.911,7.582,149.454
C05003=1127.918,73.950,-54.381,179.912,7.586,149.455
C05004=1127.912,74.200,-54.398,179.914,7.589,149.455
C05005=1127.907,74.449,-54.414,179.914,7.593,149.456
C05006=1127.902,74.699,-54.432,179.916,7.597,149.456
C05007=1127.898,74.948,-54.449,179.918,7.601,149.456
C05008=1127.893,75.163,-54.464,179.919,7.605,149.457
C05009=1127.889,75.378,-54.479,179.920,7.608,149.457
C05010=1127.885,75.593,-54.494,179.922,7.612,149.458
C05011=1127.880,75.808,-54.508,179.923,7.615,149.458
C05012=1127.876,76.023,-54.524,179.924,7.619,149.459
C05013=1127.872,76.237,-54.537,179.925,7.622,149.459
C05014=1127.868,76.452,-54.553,179.926,7.625,149.459
C05015=1127.863,76.667,-54.567,179.928,7.628,149.460
C05016=1127.859,76.917,-54.585,179.929,7.632,149.460
C05017=1127.854,77.166,-54.602,179.930,7.636,149.461
C05018=1127.849,77.416,-54.619,179.931,7.639,149.461
C05019=1127.844,77.665,-54.637,179.932,7.644,149.462
C05020=1127.839,77.915,-54.654,179.933,7.647,149.462
C05021=1127.835,78.164,-54.672,179.933,7.650,149.463
C05022=1127.829,78.413,-54.689,179.935,7.654,149.464
C05023=1127.824,78.662,-54.706,179.935,7.658,149.464
C05024=1127.819,78.912,-54.724,179.937,7.662,149.465
C05025=1127.814,79.161,-54.741,179.938,7.665,149.465
C05026=1127.809,79.410,-54.759,179.939,7.669,149.466
C05027=1127.805,79.660,-54.775,179.940,7.673,149.466
C05028=1127.800,79.909,-54.793,179.941,7.677,149.467
C05029=1127.795,80.159,-54.811,179.942,7.681,149.467
C05030=1127.790,80.408,-54.828,179.943,7.684,149.468
C05031=1127.785,80.658,-54.845,179.944,7.688,149.468
C05032=1127.780,80.907,-54.863,179.945,7.692,149.469
C05033=1127.775,81.157,-54.881,179.947,7.695,149.470
C05034=1127.770,81.405,-54.898,179.948,7.700,149.470
C05035=1127.765,81.655,-54.915,179.949,7.703,149.471
C05036=1127.760,81.904,-54.933,179.950,7.707,149.471
C05037=1127.755,82.153,-54.951,179.951,7.710,149.472
C05038=1127.751,82.402,-54.968,179.952,7.714,149.472
C05039=1127.746,82.652,-54.986,179.953,7.718,149.473
C05040=1127.741,82.901,-55.003,179.954,7.722,149.473
C05041=1127.736,83.151,-55.021,179.956,7.726,149.474
C05042=1127.731,83.400,-55.039,179.957,7.730,149.474
C05043=1127.726,83.649,-55.056,179.958,7.733,149.475
C05044=1127.721,83.898,-55.073,179.959,7.737,149.475
C05045=1127.716,84.148,-55.091,179.961,7.741,149.476
C05046=1127.711,84.397,-55.109,179.962,7.745,149.476
C05047=1127.706,84.646,-55.127,179.963,7.748,149.477
C05048=1127.701,84.896,-55.145,179.965,7.752,149.477
C05049=1127.696,85.145,-55.162,179.966,7.757,149.478
C05050=1127.692,85.394,-55.179,179.967,7.760,149.478
C05051=1127.687,85.644,-55.197,179.968,7.764,149.479
C05052=1127.682,85.893,-55.215,179.969,7.768,149.479
C05053=1127.677,86.142,-55.232,179.971,7.772,149.480
C05054=1127.672,86.392,-55.250,179.973,7.776,149.480
C05055=1127.667,86.641,-55.268,179.974,7.780,149.481
C05056=1127.662,86.890,-55.286,179.975,7.783,149.481
C05057=1127.657,87.140,-55.304,179.976,7.787,149.482
C05058=1127.652,87.389,-55.322,179.978,7.791,149.482
C05059=1127.648,87.639,-55.340,179.979,7.795,149.483
C05060=1127.643,87.888,-55.358,179.981,7.799,149.483
C05061=1127.639,88.137,-55.375,179.982,7.803,149.484
C05062=1127.634,88.387,-55.393,179.984,7.807,149.484
C05063=1127.629,88.636,-55.411,179.985,7.810,149.484
C05064=1127.624,88.851,-55.427,179.986,7.814,149.485
C05065=1127.620,89.066,-55.442,179.987,7.817,149.485
C05066=1127.616,89.280,-55.457,179.989,7.821,149.486
C05067=1127.611,89.495,-55.473,179.990,7.824,149.486
C05068=1127.607,89.710,-55.488,179.991,7.827,149.487
C05069=1127.603,89.925,-55.504,179.992,7.831,149.487
C05070=1127.599,90.139,-55.519,179.994,7.834,149.487
C05071=1127.594,90.354,-55.535,179.995,7.838,149.488
C05072=1127.590,90.604,-55.553,179.997,7.841,149.488
C05073=1127.585,90.853,-55.571,179.999,7.845,149.489
C05074=1127.580,91.103,-55.589,-180.000,7.849,149.489
C05075=1127.575,91.352,-55.607,-179.999,7.853,149.490
C05076=1127.570,91.601,-55.625,-179.997,7.857,149.490
C05077=1127.565,91.850,-55.643,-179.995,7.861,149.490
C05078=1127.560,92.099,-55.661,-179.994,7.865,149.491
C05079=1127.556,92.349,-55.679,-179.992,7.869,149.491
C05080=1127.551,92.598,-55.697,-179.991,7.873,149.492
C05081=1127.546,92.847,-55.715,-179.989,7.877,149.492
C05082=1127.541,93.097,-55.733,-179.987,7.881,149.493
C05083=1127.536,93.346,-55.751,-179.986,7.885,149.493
C05084=1127.531,93.595,-55.769,-179.984,7.889,149.493
C05085=1127.526,93.845,-55.788,-179.983,7.892,149.494
C05086=1127.522,94.094,-55.806,-179.981,7.896,149.494
C05087=1127.517,94.344,-55.824,-179.979,7.900,149.495
C05088=1127.512,94.593,-55.842,-179.977,7.904,149.495
C05089=1127.507,94.842,-55.860,-179.976,7.908,149.495
C05090=1127.503,95.091,-55.879,-179.974,7.912,149.496
C05091=1127.497,95.341,-55.898,-179.972,7.916,149.496
C05092=1127.492,95.590,-55.916,-179.970,7.920,149.497
C05093=1127.487,95.839,-55.934,-179.969,7.924,149.497
C05094=1127.482,96.088,-55.952,-179.967,7.928,149.498
C05095=1127.478,96.338,-55.970,-179.965,7.931,149.498
C05096=1127.473,96.587,-55.989,-179.963,7.936,149.498
C05097=1127.468,96.836,-56.007,-179.961,7.940,149.499
C05098=1127.463,97.085,-56.025,-179.960,7.944,149.499
C05099=1127.459,97.335,-56.044,-179.958,7.947,149.499
C05100=1127.454,97.584,-56.062,-179.956,7.951,149.500
C05101=1127.448,97.833,-56.081,-179.954,7.956,149.500
C05102=1127.444,98.083,-56.099,-179.952,7.960,149.501
C05103=1127.439,98.332,-56.117,-179.950,7.963,149.501
C05104=1127.435,98.581,-56.136,-179.949,7.967,149.501
C05105=1127.429,98.830,-56.155,-179.946,7.972,149.502
C05106=1127.425,99.080,-56.173,-179.944,7.975,149.502
C05107=1127.420,99.329,-56.192,-179.943,7.979,149.502
C05108=1127.414,99.578,-56.210,-179.941,7.983,149.503
C05109=1127.410,99.827,-56.229,-179.938,7.987,149.503
C05110=1127.405,100.077,-56.247,-179.937,7.991,149.503
C05111=1127.400,100.326,-56.266,-179.935,7.995,149.504
C05112=1127.396,100.575,-56.285,-179.932,7.999,149.504
C05113=1127.391,100.825,-56.303,-179.931,8.003,149.504
C05114=1127.385,101.073,-56.322,-179.929,8.007,149.505
C05115=1127.381,101.323,-56.341,-179.927,8.011,149.505
C05116=1127.376,101.572,-56.360,-179.925,8.015,149.505
C05117=1127.371,101.821,-56.378,-179.923,8.019,149.506
C05118=1127.367,102.071,-56.397,-179.920,8.023,149.506
C05119=1127.361,102.320,-56.415,-179.918,8.027,149.506
C05120=1127.357,102.534,-56.432,-179.917,8.031,149.507
C05121=1127.353,102.750,-56.448,-179.915,8.034,149.507
C05122=1127.349,102.964,-56.464,-179.913,8.037,149.507
C05123=1127.344,103.179,-56.480,-179.911,8.040,149.507
C05124=1127.341,103.394,-56.496,-179.909,8.044,149.508
C05125=1127.336,103.609,-56.512,-179.907,8.048,149.508
C05126=1127.333,103.823,-56.528,-179.905,8.051,149.508
C05127=1127.328,104.038,-56.544,-179.904,8.054,149.508
C05128=1127.324,104.287,-56.564,-179.901,8.058,149.508
C05129=1127.318,104.536,-56.583,-179.900,8.062,149.509
C05130=1127.314,104.786,-56.601,-179.897,8.066,149.509
C05131=1127.309,105.035,-56.620,-179.895,8.070,149.509
C05132=1127.304,105.285,-56.639,-179.892,8.074,149.510
C05133=1127.299,105.534,-56.658,-179.891,8.078,149.510
C05134=1127.295,105.783,-56.677,-179.888,8.082,149.510
C05135=1127.290,106.032,-56.696,-179.886,8.086,149.510
C05136=1127.284,106.281,-56.715,-179.884,8.089,149.511
C05137=1127.280,106.531,-56.734,-179.881,8.094,149.511
C05138=1127.275,106.779,-56.753,-179.879,8.097,149.511
C05139=1127.270,107.029,-56.772,-179.877,8.102,149.512
C05140=1127.265,107.278,-56.791,-179.874,8.106,149.512
C05141=1127.261,107.527,-56.810,-179.872,8.109,149.512
C05142=1127.256,107.776,-56.829,-179.869,8.114,149.512
C05143=1127.251,108.026,-56.849,-179.867,8.117,149.512
C05144=1127.246,108.275,-56.867,-179.865,8.122,149.513
C05145=1127.241,108.525,-56.887,-179.863,8.125,149.513
C05146=1127.236,108.773,-56.906,-179.860,8.129,149.513
C05147=1127.232,109.023,-56.925,-179.858,8.133,149.513
C05148=1127.227,109.272,-56.945,-179.855,8.137,149.514
C05149=1127.222,109.521,-56.964,-179.853,8.141,149.514
C05150=1127.218,109.770,-56.983,-179.850,8.145,149.514
C05151=1127.213,110.019,-57.002,-179.848,8.149,149.514
C05152=1127.208,110.269,-57.022,-179.846,8.153,149.514
C05153=1127.203,110.517,-57.041,-179.843,8.157,149.514
C05154=1127.198,110.767,-57.060,-179.840,8.160,149.515
C05155=1127.193,111.016,-57.079,-179.838,8.164,149.515
C05156=1127.188,111.266,-57.099,-179.836,8.168,149.515
C05157=1127.184,111.515,-57.118,-179.834,8.172,149.515
C05158=1127.179,111.764,-57.137,-179.832,8.175,149.516
C05159=1127.174,112.013,-57.157,-179.830,8.179,149.516
C05160=1127.169,112.262,-57.177,-179.828,8.182,149.516
C05161=1127.165,112.511,-57.196,-179.826,8.186,149.517
C05162=1127.160,112.761,-57.215,-179.825,8.189,149.517
C05163=1127.155,113.010,-57.235,-179.823,8.192,149.517
C05164=1127.150,113.259,-57.254,-179.821,8.196,149.517
C05165=1127.145,113.509,-57.274,-179.819,8.200,149.518
C05166=1127.141,113.757,-57.293,-179.817,8.203,149.518
C05167=1127.136,114.007,-57.312,-179.815,8.207,149.518
C05168=1127.131,114.256,-57.332,-179.813,8.210,149.518
C05169=1127.126,114.505,-57.351,-179.811,8.214,149.519
C05170=1127.121,114.754,-57.372,-179.809,8.218,149.519
C05171=1127.116,115.003,-57.391,-179.807,8.221,149.519
C05172=1127.111,115.253,-57.410,-179.805,8.225,149.519
C05173=1127.107,115.502,-57.430,-179.804,8.227,149.520
C05174=1127.102,115.751,-57.449,-179.802,8.231,149.520
C05175=1127.098,116.000,-57.469,-179.800,8.235,149.520
C05176=1127.094,116.215,-57.486,-179.798,8.238,149.521
C05177=1127.089,116.429,-57.503,-179.796,8.241,149.521
C05178=1127.085,116.644,-57.520,-179.795,8.244,149.521
C05179=1127.081,116.859,-57.537,-179.793,8.247,149.521
C05180=1127.077,117.074,-57.554,-179.792,8.250,149.521
C05181=1127.072,117.288,-57.570,-179.790,8.253,149.522
C05182=1127.068,117.503,-57.588,-179.788,8.256,149.522
C05183=1127.064,117.717,-57.605,-179.787,8.259,149.522
C05184=1127.059,117.967,-57.625,-179.785,8.262,149.522
C05185=1127.055,118.216,-57.644,-179.783,8.265,149.523
C05186=1127.051,118.465,-57.664,-179.781,8.268,149.523
C05187=1127.045,118.714,-57.683,-179.779,8.272,149.523
C05188=1127.041,118.963,-57.704,-179.777,8.276,149.523
C05189=1127.036,119.213,-57.723,-179.775,8.279,149.524
C05190=1127.031,119.462,-57.743,-179.773,8.283,149.524
C05191=1127.026,119.710,-57.763,-179.772,8.286,149.524
C05192=1127.022,119.960,-57.783,-179.770,8.289,149.524
C05193=1127.017,120.209,-57.802,-179.768,8.293,149.525
C05194=1127.012,120.458,-57.823,-179.766,8.296,149.525
C05195=1127.008,120.708,-57.842,-179.764,8.300,149.525
C05196=1127.002,120.957,-57.863,-179.763,8.303,149.525
C05197=1126.997,121.206,-57.883,-179.761,8.307,149.526
C05198=1126.993,121.455,-57.903,-179.759,8.310,149.526
C05199=1126.988,121.705,-57.923,-179.757,8.314,149.526
C05200=1126.984,121.954,-57.943,-179.755,8.316,149.526
C05201=1126.978,122.202,-57.962,-179.753,8.320,149.527
C05202=1126.974,122.451,-57.983,-179.752,8.324,149.527
C05203=1126.969,122.701,-58.002,-179.750,8.327,149.527
C05204=1126.965,122.950,-58.023,-179.748,8.330,149.528
C05205=1126.960,123.199,-58.042,-179.746,8.333,149.528
C05206=1126.955,123.448,-58.063,-179.744,8.337,149.528
C05207=1126.950,123.697,-58.082,-179.742,8.341,149.528
C05208=1126.945,123.947,-58.103,-179.741,8.343,149.529
C05209=1126.940,124.195,-58.123,-179.739,8.347,149.529
C05210=1126.936,124.445,-58.143,-179.737,8.350,149.529
C05211=1126.931,124.694,-58.163,-179.735,8.353,149.529
C05212=1126.926,124.944,-58.183,-179.734,8.357,149.530
C05213=1126.922,125.193,-58.203,-179.732,8.360,149.530
C05214=1126.916,125.441,-58.224,-179.730,8.364,149.530
C05215=1126.912,125.691,-58.244,-179.728,8.367,149.530
C05216=1126.907,125.940,-58.264,-179.727,8.371,149.531
C05217=1126.903,126.189,-58.284,-179.724,8.374,149.531
C05218=1126.898,126.438,-58.304,-179.723,8.377,149.531
C05219=1126.893,126.687,-58.325,-179.721,8.380,149.532
C05220=1126.888,126.936,-58.345,-179.719,8.384,149.532
C05221=1126.884,127.185,-58.366,-179.718,8.387,149.532
C05222=1126.879,127.435,-58.385,-179.716,8.390,149.532
C05223=1126.875,127.684,-58.406,-179.714,8.394,149.533
C05224=1126.870,127.933,-58.427,-179.713,8.397,149.533
C05225=1126.864,128.181,-58.447,-179.711,8.400,149.533
C05226=1126.860,128.431,-58.466,-179.709,8.404,149.534
C05227=1126.855,128.680,-58.487,-179.707,8.407,149.534
C05228=1126.850,128.929,-58.508,-179.706,8.411,149.534
C05229=1126.846,129.178,-58.528,-179.703,8.414,149.534
C05230=1126.841,129.428,-58.548,-179.702,8.417,149.535
C05231=1126.836,129.677,-58.569,-179.700,8.420,149.535
C05232=1126.832,129.891,-58.587,-179.699,8.423,149.535
C05233=1126.828,130.106,-58.604,-179.698,8.426,149.536
C05234=1126.823,130.321,-58.622,-179.696,8.429,149.536
C05235=1126.820,130.535,-58.639,-179.695,8.431,149.536
C05236=1126.816,130.750,-58.657,-179.693,8.434,149.536
C05237=1126.812,130.963,-58.675,-179.691,8.438,149.536
C05238=1126.807,131.179,-58.692,-179.690,8.440,149.537
C05239=1126.803,131.393,-58.710,-179.688,8.443,149.537
C05240=1126.799,131.642,-58.730,-179.687,8.446,149.537
C05241=1126.794,131.892,-58.751,-179.685,8.450,149.538
C05242=1126.789,132.140,-58.772,-179.683,8.453,149.538
C05243=1126.785,132.389,-58.792,-179.682,8.456,149.538
C05244=1126.780,132.639,-58.813,-179.680,8.460,149.538
C05245=1126.775,132.888,-58.833,-179.679,8.462,149.539
C05246=1126.770,133.137,-58.854,-179.677,8.466,149.539
C05247=1126.766,133.386,-58.875,-179.675,8.470,149.539
C05248=1126.761,133.635,-58.895,-179.673,8.473,149.540
C05249=1126.756,133.884,-58.916,-179.672,8.476,149.540
C05250=1126.751,134.133,-58.936,-179.670,8.479,149.540
C05251=1126.746,134.382,-58.957,-179.668,8.483,149.540
C05252=1126.742,134.631,-58.978,-179.667,8.486,149.541
C05253=1126.737,134.880,-58.999,-179.665,8.489,149.541
C05254=1126.732,135.129,-59.019,-179.664,8.493,149.541
C05255=1126.727,135.379,-59.040,-179.662,8.496,149.542
C05256=1126.723,135.628,-59.061,-179.660,8.499,149.542
C05257=1126.718,135.878,-59.082,-179.659,8.502,149.542
C05258=1126.714,136.127,-59.102,-179.657,8.506,149.543
C05259=1126.708,136.376,-59.123,-179.656,8.509,149.543
C05260=1126.704,136.624,-59.144,-179.654,8.512,149.543
C05261=1126.699,136.873,-59.165,-179.652,8.515,149.543
C05262=1126.695,137.122,-59.186,-179.651,8.519,149.544
C05263=1126.690,137.372,-59.207,-179.649,8.522,149.544
C05264=1126.685,137.621,-59.227,-179.648,8.526,149.545
C05265=1126.680,137.870,-59.248,-179.646,8.529,149.545
C05266=1126.676,138.119,-59.268,-179.645,8.532,149.545
C05267=1126.671,138.368,-59.290,-179.643,8.536,149.545
C05268=1126.667,138.617,-59.311,-179.642,8.539,149.546
C05269=1126.662,138.866,-59.332,-179.639,8.542,149.546
C05270=1126.656,139.116,-59.353,-179.638,8.545,149.546
C05271=1126.652,139.364,-59.374,-179.636,8.549,149.547
C05272=1126.647,139.613,-59.395,-179.635,8.552,149.547
C05273=1126.643,139.862,-59.415,-179.633,8.555,149.547
C05274=1126.638,140.112,-59.436,-179.632,8.558,149.548
C05275=1126.634,140.360,-59.457,-179.630,8.562,149.548
C05276=1126.629,140.610,-59.478,-179.629,8.565,149.549
C05277=1126.624,140.859,-59.499,-179.627,8.569,149.549
C05278=1126.620,141.107,-59.521,-179.626,8.572,149.549
C05279=1126.614,141.356,-59.541,-179.624,8.575,149.549
C05280=1126.610,141.606,-59.563,-179.623,8.578,149.550
C05281=1126.606,141.855,-59.584,-179.621,8.582,149.550
C05282=1126.600,142.104,-59.605,-179.620,8.585,149.551
C05283=1126.595,142.353,-59.626,-179.618,8.588,149.551
C05284=1126.591,142.602,-59.647,-179.617,8.591,149.551
C05285=1126.586,142.851,-59.668,-179.615,8.595,149.552
C05286=1126.581,143.101,-59.689,-179.614,8.598,149.552
C05287=1126.577,143.349,-59.710,-179.612,8.602,149.552
C05288=1126.573,143.564,-59.729,-179.611,8.605,149.552
C05289=1126.569,143.778,-59.746,-179.610,8.607,149.553
C05290=1126.565,143.993,-59.766,-179.609,8.610,149.553
C05291=1126.561,144.207,-59.784,-179.607,8.612,149.553
C05292=1126.557,144.422,-59.802,-179.606,8.615,149.554
C05293=1126.552,144.636,-59.820,-179.605,8.618,149.554
C05294=1126.549,144.850,-59.838,-179.604,8.621,149.554
C05295=1126.544,145.065,-59.857,-179.602,8.624,149.555
C05296=1126.540,145.315,-59.878,-179.600,8.628,149.555
C05297=1126.536,145.563,-59.899,-179.597,8.632,149.555
C05298=1126.531,145.812,-59.920,-179.594,8.637,149.555
C05299=1126.526,146.061,-59.942,-179.592,8.640,149.555
C05300=1126.521,146.311,-59.963,-179.589,8.644,149.556
C05301=1126.516,146.560,-59.985,-179.586,8.648,149.556
C05302=1126.512,146.809,-60.005,-179.584,8.652,149.556
C05303=1126.507,147.057,-60.027,-179.581,8.656,149.556
C05304=1126.503,147.306,-60.049,-179.578,8.660,149.556
C05305=1126.497,147.556,-60.070,-179.576,8.664,149.557
C05306=1126.493,147.804,-60.091,-179.574,8.668,149.557
C05307=1126.488,148.054,-60.113,-179.571,8.671,149.557
C05308=1126.484,148.303,-60.134,-179.568,8.675,149.557
C05309=1126.479,148.551,-60.155,-179.566,8.679,149.557
C05310=1126.475,148.801,-60.178,-179.563,8.683,149.557
C05311=1126.470,149.050,-60.199,-179.560,8.687,149.558
C05312=1126.465,149.299,-60.220,-179.558,8.690,149.558
C05313=1126.460,149.548,-60.242,-179.555,8.694,149.558
C05314=1126.455,149.797,-60.263,-179.553,8.698,149.558
C05315=1126.450,150.046,-60.285,-179.550,8.702,149.558
C05316=1126.446,150.295,-60.307,-179.548,8.705,149.558
C05317=1126.441,150.544,-60.329,-179.545,8.709,149.559
C05318=1126.436,150.792,-60.350,-179.543,8.713,149.559
C05319=1126.432,151.042,-60.372,-179.540,8.717,149.559
C05320=1126.427,151.291,-60.393,-179.538,8.720,149.559
C05321=1126.423,151.540,-60.415,-179.535,8.724,149.559
C05322=1126.418,151.789,-60.437,-179.533,8.728,149.559
C05323=1126.413,152.038,-60.459,-179.529,8.731,149.559
C05324=1126.409,152.287,-60.481,-179.527,8.735,149.560
C05325=1126.404,152.536,-60.502,-179.525,8.739,149.560
C05326=1126.400,152.785,-60.525,-179.522,8.742,149.560
C05327=1126.394,153.034,-60.545,-179.520,8.746,149.560
C05328=1126.389,153.283,-60.567,-179.517,8.750,149.560
C05329=1126.385,153.532,-60.589,-179.515,8.753,149.560
C05330=1126.380,153.781,-60.611,-179.512,8.757,149.560
C05331=1126.376,154.030,-60.633,-179.510,8.760,149.561
C05332=1126.371,154.279,-60.655,-179.507,8.764,149.561
C05333=1126.367,154.528,-60.677,-179.504,8.768,149.561
C05334=1126.362,154.777,-60.698,-179.502,8.771,149.561
C05335=1126.357,155.026,-60.721,-179.500,8.774,149.561
C05336=1126.352,155.275,-60.743,-179.497,8.778,149.561
C05337=1126.348,155.524,-60.765,-179.494,8.781,149.561
C05338=1126.343,155.772,-60.787,-179.492,8.785,149.561
C05339=1126.339,156.022,-60.809,-179.489,8.788,149.562
C05340=1126.334,156.270,-60.831,-179.487,8.792,149.562
C05341=1126.329,156.520,-60.853,-179.484,8.795,149.562
C05342=1126.324,156.769,-60.875,-179.482,8.799,149.562
C05343=1126.320,157.018,-60.897,-179.480,8.802,149.562
C05344=1126.316,157.232,-60.916,-179.477,8.805,149.562
C05345=1126.312,157.446,-60.935,-179.475,8.809,149.562
C05346=1126.308,157.661,-60.954,-179.473,8.811,149.562
C05347=1126.304,157.875,-60.974,-179.471,8.814,149.562
C05348=1126.300,158.090,-60.993,-179.469,8.818,149.563
C05349=1126.296,158.304,-61.012,-179.467,8.820,149.563
C05350=1126.292,158.518,-61.031,-179.464,8.823,149.563
C05351=1126.288,158.733,-61.050,-179.463,8.826,149.563
C05352=1126.284,158.982,-61.072,-179.460,8.830,149.563
C05353=1126.279,159.230,-61.094,-179.457,8.833,149.563
C05354=1126.274,159.480,-61.117,-179.455,8.836,149.563
C05355=1126.269,159.728,-61.139,-179.452,8.839,149.563
C05356=1126.265,159.977,-61.161,-179.450,8.842,149.563
C05357=1126.261,160.227,-61.183,-179.448,8.846,149.563
C05358=1126.255,160.475,-61.206,-179.445,8.849,149.563
C05359=1126.251,160.724,-61.228,-179.442,8.853,149.564
C05360=1126.247,160.974,-61.250,-179.440,8.856,149.564
C05361=1126.242,161.222,-61.273,-179.438,8.859,149.564
C05362=1126.237,161.471,-61.295,-179.435,8.863,149.564
C05363=1126.232,161.720,-61.317,-179.433,8.866,149.564
C05364=1126.228,161.969,-61.340,-179.430,8.869,149.564
C05365=1126.224,162.218,-61.362,-179.428,8.872,149.564
C05366=1126.218,162.467,-61.385,-179.426,8.876,149.564
C05367=1126.214,162.716,-61.407,-179.423,8.879,149.564
C05368=1126.210,162.965,-61.430,-179.421,8.882,149.564
C05369=1126.204,163.214,-61.452,-179.419,8.885,149.565
C05370=1126.200,163.462,-61.475,-179.416,8.889,149.565
C05371=1126.195,163.712,-61.498,-179.414,8.892,149.565
C05372=1126.191,163.960,-61.520,-179.411,8.895,149.565
C05373=1126.187,164.209,-61.542,-179.409,8.898,149.565
C05374=1126.182,164.458,-61.566,-179.406,8.901,149.565
C05375=1126.178,164.708,-61.588,-179.404,8.904,149.565
C05376=1126.172,164.956,-61.611,-179.402,8.908,149.565
C05377=1126.168,165.205,-61.633,-179.399,8.911,149.565
C05378=1126.163,165.454,-61.656,-179.397,8.914,149.565
C05379=1126.159,165.703,-61.679,-179.394,8.917,149.565
C05380=1126.154,165.952,-61.701,-179.392,8.921,149.566
C05381=1126.150,166.201,-61.724,-179.390,8.924,149.566
C05382=1126.145,166.451,-61.747,-179.387,8.927,149.566
C05383=1126.140,166.699,-61.769,-179.385,8.930,149.566
C05384=1126.136,166.948,-61.792,-179.383,8.934,149.566
C05385=1126.131,167.197,-61.814,-179.380,8.937,149.566
C05386=1126.127,167.446,-61.838,-179.377,8.940,149.566
C05387=1126.121,167.694,-61.861,-179.376,8.942,149.566
C05388=1126.117,167.943,-61.883,-179.373,8.946,149.566
C05389=1126.112,168.193,-61.906,-179.371,8.949,149.566
C05390=1126.108,168.441,-61.929,-179.368,8.952,149.566
C05391=1126.103,168.690,-61.952,-179.366,8.955,149.567
C05392=1126.098,168.939,-61.975,-179.364,8.958,149.567
C05393=1126.094,169.188,-61.997,-179.361,8.962,149.567
C05394=1126.089,169.437,-62.021,-179.359,8.964,149.567
C05395=1126.085,169.686,-62.043,-179.357,8.967,149.567
C05396=1126.080,169.934,-62.066,-179.355,8.970,149.567
C05397=1126.075,170.184,-62.089,-179.352,8.974,149.567
C05398=1126.071,170.433,-62.112,-179.350,8.977,149.567
C05399=1126.066,170.682,-62.135,-179.348,8.980,149.567
C05400=1126.063,170.895,-62.155,-179.346,8.982,149.567
C05401=1126.058,171.110,-62.175,-179.344,8.985,149.567
C05402=1126.055,171.324,-62.195,-179.342,8.987,149.567
C05403=1126.050,171.538,-62.215,-179.340,8.991,149.568
C05404=1126.047,171.753,-62.235,-179.338,8.993,149.568
C05405=1126.043,171.967,-62.254,-179.336,8.995,149.568
C05406=1126.039,172.181,-62.275,-179.334,8.998,149.568
C05407=1126.035,172.396,-62.294,-179.332,9.001,149.568
C05408=1126.030,172.645,-62.317,-179.330,9.003,149.568
C05409=1126.025,172.894,-62.340,-179.328,9.007,149.568
C05410=1126.021,173.142,-62.363,-179.325,9.010,149.568
C05411=1126.017,173.391,-62.386,-179.324,9.012,149.568
C05412=1126.011,173.640,-62.409,-179.321,9.015,149.568
C05413=1126.007,173.889,-62.433,-179.319,9.019,149.568
C05414=1126.003,174.138,-62.456,-179.317,9.022,149.569
C05415=1125.998,174.387,-62.479,-179.315,9.024,149.569
C05416=1125.993,174.636,-62.502,-179.312,9.027,149.569
C05417=1125.988,174.885,-62.526,-179.310,9.031,149.569
C05418=1125.984,175.133,-62.550,-179.308,9.033,149.569
C05419=1125.980,175.382,-62.572,-179.306,9.036,149.569
C05420=1125.975,175.631,-62.596,-179.303,9.039,149.569
C05421=1125.971,175.880,-62.619,-179.302,9.042,149.569
C05422=1125.966,176.129,-62.643,-179.299,9.045,149.569
C05423=1125.961,176.378,-62.666,-179.297,9.048,149.569
C05424=1125.957,176.626,-62.688,-179.295,9.051,149.570
C05425=1125.952,176.875,-62.712,-179.293,9.054,149.570
C05426=1125.947,177.124,-62.735,-179.290,9.057,149.570
C05427=1125.943,177.372,-62.759,-179.289,9.060,149.570
C05428=1125.938,177.621,-62.782,-179.286,9.063,149.570
C05429=1125.934,177.870,-62.806,-179.284,9.066,149.570
C05430=1125.929,178.120,-62.829,-179.282,9.069,149.570
C05431=1125.924,178.369,-62.853,-179.280,9.072,149.570
C05432=1125.920,178.617,-62.876,-179.278,9.074,149.570
C05433=1125.916,178.866,-62.899,-179.276,9.078,149.570
C05434=1125.911,179.115,-62.923,-179.273,9.081,149.571
C05435=1125.906,179.364,-62.946,-179.271,9.084,149.571
C05436=1125.902,179.612,-62.970,-179.268,9.087,149.571
C05437=1125.897,179.861,-62.994,-179.265,9.091,149.571
C05438=1125.893,180.110,-63.017,-179.262,9.094,149.571
C05439=1125.888,180.359,-63.041,-179.259,9.098,149.571
C05440=1125.884,180.608,-63.064,-179.256,9.101,149.571
C05441=1125.879,180.857,-63.088,-179.254,9.104,149.571
C05442=1125.874,181.105,-63.112,-179.250,9.107,149.570
C05443=1125.870,181.355,-63.135,-179.248,9.111,149.571
C05444=1125.866,181.604,-63.159,-179.245,9.114,149.571
C05445=1125.861,181.852,-63.183,-179.242,9.118,149.571
C05446=1125.857,182.101,-63.206,-179.239,9.120,149.570
C05447=1125.852,182.350,-63.230,-179.236,9.123,149.571
C05448=1125.847,182.599,-63.254,-179.234,9.126,149.571
C05449=1125.843,182.847,-63.278,-179.231,9.130,149.571
C05450=1125.838,183.096,-63.301,-179.228,9.133,149.570
C05451=1125.834,183.345,-63.325,-179.225,9.136,149.570
C05452=1125.829,183.594,-63.349,-179.223,9.139,149.571
C05453=1125.824,183.842,-63.373,-179.220,9.142,149.571
C05454=1125.820,184.092,-63.397,-179.217,9.145,149.570
C05455=1125.816,184.341,-63.421,-179.215,9.148,149.570
C05456=1125.811,184.554,-63.441,-179.213,9.151,149.570
C05457=1125.808,184.769,-63.462,-179.210,9.154,149.571
C05458=1125.803,184.983,-63.482,-179.208,9.156,149.571
C05459=1125.799,185.197,-63.503,-179.206,9.159,149.571
C05460=1125.796,185.412,-63.524,-179.204,9.161,149.570
C05461=1125.792,185.625,-63.544,-179.202,9.163,149.570
C05462=1125.788,185.839,-63.565,-179.199,9.167,149.571
C05463=1125.784,186.054,-63.586,-179.197,9.169,149.571
C05464=1125.780,186.302,-63.610,-179.195,9.172,149.571
C05465=1125.775,186.551,-63.633,-179.192,9.175,149.571
C05466=1125.771,186.800,-63.657,-179.190,9.177,149.571
C05467=1125.766,187.048,-63.682,-179.188,9.181,149.571
C05468=1125.761,187.297,-63.705,-179.185,9.184,149.571
C05469=1125.757,187.547,-63.730,-179.183,9.186,149.571
C05470=1125.753,187.795,-63.754,-179.180,9.189,149.571
C05471=1125.747,188.044,-63.778,-179.178,9.192,149.571
C05472=1125.743,188.293,-63.802,-179.176,9.194,149.571
C05473=1125.739,188.541,-63.826,-179.174,9.197,149.571
C05474=1125.735,188.790,-63.850,-179.171,9.200,149.571
C05475=1125.730,189.039,-63.875,-179.169,9.203,149.571
C05476=1125.725,189.288,-63.898,-179.167,9.206,149.571
C05477=1125.721,189.536,-63.922,-179.165,9.208,149.571
C05478=1125.716,189.786,-63.947,-179.163,9.212,149.571
C05479=1125.712,190.034,-63.971,-179.161,9.214,149.571
C05480=1125.707,190.283,-63.995,-179.158,9.217,149.571
C05481=1125.702,190.532,-64.019,-179.156,9.219,149.571
C05482=1125.697,190.780,-64.043,-179.154,9.222,149.571
C05483=1125.694,191.030,-64.068,-179.152,9.225,149.571
C05484=1125.688,191.278,-64.093,-179.150,9.227,149.571
C05485=1125.684,191.527,-64.117,-179.148,9.230,149.572
C05486=1125.680,191.775,-64.141,-179.146,9.233,149.572
